LIN {X 0,Y 572.94,Z 558.785,A -85,B 0,C 180,E1 -2249.297,E2 -2249.297} C_VEL
LIN {X 0,Y 572.938,Z 559,A -85,B 0,C 180,E1 -2250,E2 -2250} C_VEL
LIN {X 0,Y 572.946,Z 558.187,A -85,B 0,C 180,E1 -2251.405,E2 -2251.405} C_VEL
LIN {X 0,Y 572.938,Z 557.2,A -85,B 0,C 180,E1 -2252.109,E2 -2252.109} C_VEL
LIN {X 0,Y 572.959,Z 555.811,A -85,B 0,C 180,E1 -2252.812,E2 -2252.812} C_VEL
LIN {X 0,Y 573.014,Z 552.897,A -85,B 0,C 180,E1 -2253.868,E2 -2253.868} C_VEL
LIN {X 0,Y 572.963,Z 548.951,A -85,B 0,C 180,E1 -2254.925,E2 -2254.925} C_VEL
LIN {X 0,Y 573.068,Z 542.879,A -85,B 0,C 180,E1 -2256.16,E2 -2256.16} C_VEL
LIN {X 0,Y 573.119,Z 536.241,A -85,B 0,C 180,E1 -2257.22,E2 -2257.22} C_VEL
LIN {X 0,Y 573.192,Z 527.995,A -85,B 0,C 180,E1 -2258.283,E2 -2258.283} C_VEL
LIN {X 0,Y 573.319,Z 517.606,A -85,B 0,C 180,E1 -2259.347,E2 -2259.347} C_VEL
LIN {X 0,Y 573.43,Z 507.931,A -85,B 0,C 180,E1 -2260.147,E2 -2260.147} C_VEL
LIN {X 0,Y 573.549,Z 497.409,A -85,B 0,C 180,E1 -2260.854,E2 -2260.854} C_VEL
LIN {X 0,Y 573.652,Z 486.295,A -85,B 0,C 180,E1 -2261.447,E2 -2261.447} C_VEL
LIN {X 0,Y 573.719,Z 473.186,A -85,B 0,C 180,E1 -2261.974,E2 -2261.974} C_VEL
LIN {X 0,Y 573.813,Z 460.539,A -85,B 0,C 180,E1 -2262.331,E2 -2262.331} C_VEL
LIN {X 0,Y 573.908,Z 447.35,A -85,B 0,C 180,E1 -2262.554,E2 -2262.554} C_VEL
LIN {X 0,Y 573.909,Z 350.315,A -85,B 0,C 180,E1 -2263.775,E2 -2263.775} C_VEL
LIN {X 0,Y 573.398,Z 346.617,A -85,B 0,C 180,E1 -2263.85,E2 -2263.85} C_VEL
LIN {X 0,Y 573.568,Z 326.123,A -85,B 0,C 180,E1 -2266.727,E2 -2266.727} C_VEL
LIN {X 0,Y 573.802,Z 305.615,A -85,B 0,C 180,E1 -2269.646,E2 -2269.646} C_VEL
LIN {X 0,Y 574.043,Z 285.799,A -85,B 0,C 180,E1 -2272.494,E2 -2272.494} C_VEL
LIN {X 0,Y 573.587,Z 280.858,A -85,B 0,C 180,E1 -2273.226,E2 -2273.226} C_VEL
LIN {X 0,Y 573.268,Z 279.079,A -85,B 0,C 180,E1 -2273.519,E2 -2273.519} C_VEL
LIN {X 0,Y 573.26,Z 279.079,A -85,B 0,C 180,E1 -2276.189,E2 -2276.189} C_VEL
LIN {X 0,Y 573.238,Z 279.076,A -85,B 0,C 180,E1 -2278.564,E2 -2278.564} C_VEL
LIN {X 0,Y 573.225,Z 279.075,A -85,B 0,C 180,E1 -2280.993,E2 -2280.993} C_VEL
LIN {X 0,Y 573.261,Z 279.072,A -85,B 0,C 180,E1 -2283.523,E2 -2283.523} C_VEL
LIN {X 0,Y 573.212,Z 279.084,A -85,B 0,C 180,E1 -2286.051,E2 -2286.051} C_VEL
LIN {X 0,Y 573.239,Z 279.077,A -85,B 0,C 180,E1 -2288.701,E2 -2288.701} C_VEL
LIN {X 0,Y 573.251,Z 279.072,A -85,B 0,C 180,E1 -2291.595,E2 -2291.595} C_VEL
LIN {X 0,Y 573.232,Z 279.082,A -85,B 0,C 180,E1 -2294.333,E2 -2294.333} C_VEL
LIN {X 0,Y 573.237,Z 279.074,A -85,B 0,C 180,E1 -2297.358,E2 -2297.358} C_VEL
LIN {X 0,Y 573.243,Z 279.079,A -85,B 0,C 180,E1 -2300.392,E2 -2300.392} C_VEL
LIN {X 0,Y 573.252,Z 279.076,A -85,B 0,C 180,E1 -2303.077,E2 -2303.077} C_VEL
LIN {X 0,Y 573.263,Z 279.07,A -85,B 0,C 180,E1 -2305.671,E2 -2305.671} C_VEL
LIN {X 0,Y 573.244,Z 279.074,A -85,B 0,C 180,E1 -2308.185,E2 -2308.185} C_VEL
LIN {X 0,Y 573.26,Z 279.076,A -85,B 0,C 180,E1 -2310.634,E2 -2310.634} C_VEL
LIN {X 0,Y 573.247,Z 279.083,A -85,B 0,C 180,E1 -2313.024,E2 -2313.024} C_VEL
LIN {X 0,Y 573.27,Z 279.075,A -85,B 0,C 180,E1 -2315.366,E2 -2315.366} C_VEL
LIN {X 0,Y 573.222,Z 279.076,A -85,B 0,C 180,E1 -2318.419,E2 -2318.419} C_VEL
LIN {X 0,Y 573.272,Z 279.072,A -85,B 0,C 180,E1 -2320.728,E2 -2320.728} C_VEL
LIN {X 0,Y 573.244,Z 279.077,A -85,B 0,C 180,E1 -2323.622,E2 -2323.622} C_VEL
LIN {X 0,Y 573.266,Z 279.073,A -85,B 0,C 180,E1 -2325.807,E2 -2325.807} C_VEL
LIN {X 0,Y 573.256,Z 279.072,A -85,B 0,C 180,E1 -2328.745,E2 -2328.745} C_VEL
LIN {X 0,Y 573.283,Z 279.078,A -85,B 0,C 180,E1 -2331.541,E2 -2331.541} C_VEL
LIN {X 0,Y 573.283,Z 279.068,A -85,B 0,C 180,E1 -2334.372,E2 -2334.372} C_VEL
LIN {X 0,Y 573.297,Z 279.073,A -85,B 0,C 180,E1 -2337.893,E2 -2337.893} C_VEL
LIN {X 0,Y 573.321,Z 279.063,A -85,B 0,C 180,E1 -2340.703,E2 -2340.703} C_VEL
LIN {X 0,Y 573.238,Z 279.079,A -85,B 0,C 180,E1 -2343.515,E2 -2343.515} C_VEL
LIN {X 0,Y 573.289,Z 279.073,A -85,B 0,C 180,E1 -2345.628,E2 -2345.628} C_VEL
LIN {X 0,Y 573.277,Z 279.071,A -85,B 0,C 180,E1 -2348.46,E2 -2348.46} C_VEL
LIN {X 0,Y 573.266,Z 279.071,A -85,B 0,C 180,E1 -2351.312,E2 -2351.312} C_VEL
LIN {X 0,Y 573.253,Z 279.081,A -85,B 0,C 180,E1 -2354.194,E2 -2354.194} C_VEL
LIN {X 0,Y 573.252,Z 279.072,A -85,B 0,C 180,E1 -2357.112,E2 -2357.112} C_VEL
LIN {X 0,Y 573.236,Z 279.081,A -85,B 0,C 180,E1 -2360.078,E2 -2360.078} C_VEL
LIN {X 0,Y 573.228,Z 279.086,A -85,B 0,C 180,E1 -2362.338,E2 -2362.338} C_VEL
LIN {X 0,Y 573.241,Z 279.077,A -85,B 0,C 180,E1 -2364.37,E2 -2364.37} C_VEL
LIN {X 0,Y 572.61,Z 279.158,A -85,B 0,C 180,E1 -2364.956,E2 -2364.956} C_VEL
LIN {X 0,Y 569.752,Z 279.513,A -85,B 0,C 180,E1 -2365.907,E2 -2365.907} C_VEL
LIN {X 0,Y 567.308,Z 279.819,A -85,B 0,C 180,E1 -2366.673,E2 -2366.673} C_VEL
LIN {X 0,Y 566.252,Z 279.944,A -85,B 0,C 180,E1 -2367.264,E2 -2367.264} C_VEL
LIN {X 0,Y 566.163,Z 279.955,A -85,B 0,C 180,E1 -2367.464,E2 -2367.464} C_VEL
LIN {X 0,Y 566.195,Z 279.951,A -85,B 0,C 180,E1 -2369.77,E2 -2369.77} C_VEL
LIN {X 0,Y 566.2,Z 279.958,A -85,B 0,C 180,E1 -2372.431,E2 -2372.431} C_VEL
LIN {X 0,Y 566.175,Z 279.958,A -85,B 0,C 180,E1 -2374.99,E2 -2374.99} C_VEL
LIN {X 0,Y 566.192,Z 279.952,A -85,B 0,C 180,E1 -2377.462,E2 -2377.462} C_VEL
LIN {X 0,Y 566.203,Z 279.951,A -85,B 0,C 180,E1 -2380.2,E2 -2380.2} C_VEL
LIN {X 0,Y 566.186,Z 279.96,A -85,B 0,C 180,E1 -2383.056,E2 -2383.056} C_VEL
LIN {X 0,Y 566.191,Z 279.951,A -85,B 0,C 180,E1 -2386.05,E2 -2386.05} C_VEL
LIN {X 0,Y 566.201,Z 279.958,A -85,B 0,C 180,E1 -2389.216,E2 -2389.216} C_VEL
LIN {X 0,Y 566.178,Z 279.956,A -85,B 0,C 180,E1 -2391.637,E2 -2391.637} C_VEL
LIN {X 0,Y 566.149,Z 279.956,A -85,B 0,C 180,E1 -2394.308,E2 -2394.308} C_VEL
LIN {X 0,Y 566.195,Z 279.955,A -85,B 0,C 180,E1 -2396.897,E2 -2396.897} C_VEL
LIN {X 0,Y 566.163,Z 279.964,A -85,B 0,C 180,E1 -2399.407,E2 -2399.407} C_VEL
LIN {X 0,Y 566.171,Z 279.957,A -85,B 0,C 180,E1 -2401.856,E2 -2401.856} C_VEL
LIN {X 0,Y 566.174,Z 279.954,A -85,B 0,C 180,E1 -2404.25,E2 -2404.25} C_VEL
LIN {X 0,Y 566.176,Z 279.96,A -85,B 0,C 180,E1 -2407.369,E2 -2407.369} C_VEL
LIN {X 0,Y 566.205,Z 279.96,A -85,B 0,C 180,E1 -2409.663,E2 -2409.663} C_VEL
LIN {X 0,Y 566.198,Z 279.951,A -85,B 0,C 180,E1 -2412.898,E2 -2412.898} C_VEL
LIN {X 0,Y 566.232,Z 279.954,A -85,B 0,C 180,E1 -2415.627,E2 -2415.627} C_VEL
LIN {X 0,Y 566.194,Z 279.951,A -85,B 0,C 180,E1 -2418.7,E2 -2418.7} C_VEL
LIN {X 0,Y 566.19,Z 279.954,A -85,B 0,C 180,E1 -2421.434,E2 -2421.434} C_VEL
LIN {X 0,Y 566.234,Z 279.952,A -85,B 0,C 180,E1 -2424.302,E2 -2424.302} C_VEL
LIN {X 0,Y 566.279,Z 279.947,A -85,B 0,C 180,E1 -2427.867,E2 -2427.867} C_VEL
LIN {X 0,Y 566.288,Z 279.947,A -85,B 0,C 180,E1 -2430,E2 -2430} C_VEL
LIN {X 0,Y 566.24,Z 279.947,A -85,B 0,C 180,E1 -2432.846,E2 -2432.846} C_VEL
LIN {X 0,Y 566.224,Z 279.948,A -85,B 0,C 180,E1 -2435.699,E2 -2435.699} C_VEL
LIN {X 0,Y 566.185,Z 279.96,A -85,B 0,C 180,E1 -2438.567,E2 -2438.567} C_VEL
LIN {X 0,Y 566.162,Z 279.955,A -85,B 0,C 180,E1 -2441.456,E2 -2441.456} C_VEL
LIN {X 0,Y 566.18,Z 279.962,A -85,B 0,C 180,E1 -2444.482,E2 -2444.482} C_VEL
LIN {X 0,Y 566.173,Z 279.954,A -85,B 0,C 180,E1 -2447.333,E2 -2447.333} C_VEL
LIN {X 0,Y 566.175,Z 279.953,A -85,B 0,C 180,E1 -2449.582,E2 -2449.582} C_VEL
LIN {X 0,Y 566.151,Z 279.957,A -85,B 0,C 180,E1 -2451.865,E2 -2451.865} C_VEL
LIN {X 0,Y 566.145,Z 279.96,A -85,B 0,C 180,E1 -2454.183,E2 -2454.183} C_VEL
LIN {X 0,Y 566.152,Z 279.964,A -85,B 0,C 180,E1 -2456.647,E2 -2456.647} C_VEL
LIN {X 0,Y 566.155,Z 279.966,A -85,B 0,C 180,E1 -2457.844,E2 -2457.844} C_VEL
LIN {X 0,Y 566.475,Z 284.764,A -85,B 0,C 180,E1 -2458.741,E2 -2458.741} C_VEL
LIN {X 0,Y 566.312,Z 299.374,A -85,B 0,C 180,E1 -2461.415,E2 -2461.415} C_VEL
LIN {X 0,Y 566.197,Z 308.432,A -85,B 0,C 180,E1 -2463.054,E2 -2463.054} C_VEL
LIN {X 0,Y 567.12,Z 313.95,A -85,B 0,C 180,E1 -2463.148,E2 -2463.148} C_VEL
LIN {X 0,Y 566.975,Z 415.264,A -85,B 0,C 180,E1 -2464.454,E2 -2464.454} C_VEL
LIN {X 0,Y 566.835,Z 428.571,A -85,B 0,C 180,E1 -2464.774,E2 -2464.774} C_VEL
LIN {X 0,Y 566.731,Z 439.996,A -85,B 0,C 180,E1 -2465.181,E2 -2465.181} C_VEL
LIN {X 0,Y 566.598,Z 450.313,A -85,B 0,C 180,E1 -2465.661,E2 -2465.661} C_VEL
LIN {X 0,Y 566.503,Z 460.478,A -85,B 0,C 180,E1 -2466.255,E2 -2466.255} C_VEL
LIN {X 0,Y 566.359,Z 469.422,A -85,B 0,C 180,E1 -2466.891,E2 -2466.891} C_VEL
LIN {X 0,Y 566.251,Z 477.431,A -85,B 0,C 180,E1 -2467.569,E2 -2467.569} C_VEL
LIN {X 0,Y 566.164,Z 485.34,A -85,B 0,C 180,E1 -2468.365,E2 -2468.365} C_VEL
LIN {X 0,Y 566.068,Z 492.963,A -85,B 0,C 180,E1 -2469.286,E2 -2469.286} C_VEL
LIN {X 0,Y 565.979,Z 499.365,A -85,B 0,C 180,E1 -2470.219,E2 -2470.219} C_VEL
LIN {X 0,Y 565.956,Z 504.694,A -85,B 0,C 180,E1 -2471.159,E2 -2471.159} C_VEL
LIN {X 0,Y 565.94,Z 509.114,A -85,B 0,C 180,E1 -2472.113,E2 -2472.113} C_VEL
LIN {X 0,Y 565.897,Z 512.699,A -85,B 0,C 180,E1 -2473.083,E2 -2473.083} C_VEL
LIN {X 0,Y 565.874,Z 515.471,A -85,B 0,C 180,E1 -2474.068,E2 -2474.068} C_VEL
LIN {X 0,Y 565.845,Z 517.452,A -85,B 0,C 180,E1 -2475.069,E2 -2475.069} C_VEL
LIN {X 0,Y 565.854,Z 518.623,A -85,B 0,C 180,E1 -2476.085,E2 -2476.085} C_VEL
LIN {X 0,Y 565.861,Z 518.99,A -85,B 0,C 180,E1 -2477.12,E2 -2477.12} C_VEL
LIN {X 0,Y 565.863,Z 518.499,A -85,B 0,C 180,E1 -2478.176,E2 -2478.176} C_VEL
LIN {X 0,Y 565.839,Z 517.081,A -85,B 0,C 180,E1 -2479.258,E2 -2479.258} C_VEL
LIN {X 0,Y 565.864,Z 513.657,A -85,B 0,C 180,E1 -2480.697,E2 -2480.697} C_VEL
LIN {X 0,Y 565.914,Z 510.584,A -85,B 0,C 180,E1 -2481.615,E2 -2481.615} C_VEL
LIN {X 0,Y 565.941,Z 506.208,A -85,B 0,C 180,E1 -2482.633,E2 -2482.633} C_VEL
LIN {X 0,Y 566.015,Z 500.789,A -85,B 0,C 180,E1 -2483.642,E2 -2483.642} C_VEL
LIN {X 0,Y 566.035,Z 493.84,A -85,B 0,C 180,E1 -2484.687,E2 -2484.687} C_VEL
LIN {X 0,Y 566.147,Z 486.369,A -85,B 0,C 180,E1 -2485.609,E2 -2485.609} C_VEL
LIN {X 0,Y 566.267,Z 477.878,A -85,B 0,C 180,E1 -2486.479,E2 -2486.479} C_VEL
LIN {X 0,Y 566.346,Z 468.29,A -85,B 0,C 180,E1 -2487.289,E2 -2487.289} C_VEL
LIN {X 0,Y 566.531,Z 456.725,A -85,B 0,C 180,E1 -2488.077,E2 -2488.077} C_VEL
LIN {X 0,Y 566.659,Z 445.1,A -85,B 0,C 180,E1 -2488.689,E2 -2488.689} C_VEL
LIN {X 0,Y 566.783,Z 433.171,A -85,B 0,C 180,E1 -2489.164,E2 -2489.164} C_VEL
LIN {X 0,Y 566.838,Z 422.732,A -85,B 0,C 180,E1 -2489.472,E2 -2489.472} C_VEL
LIN {X 0,Y 566.928,Z 410.787,A -85,B 0,C 180,E1 -2489.708,E2 -2489.708} C_VEL
LIN {X 0,Y 567.115,Z 313.681,A -85,B 0,C 180,E1 -2490.946,E2 -2490.946} C_VEL
LIN {X 0,Y 566.181,Z 308.374,A -85,B 0,C 180,E1 -2491.046,E2 -2491.046} C_VEL
LIN {X 0,Y 566.333,Z 295.048,A -85,B 0,C 180,E1 -2493.464,E2 -2493.464} C_VEL
LIN {X 0,Y 566.44,Z 282.076,A -85,B 0,C 180,E1 -2495.83,E2 -2495.83} C_VEL
LIN {X 0,Y 566.233,Z 279.951,A -85,B 0,C 180,E1 -2496.21,E2 -2496.21} C_VEL
LIN {X 0,Y 566.211,Z 279.955,A -85,B 0,C 180,E1 -2498.902,E2 -2498.902} C_VEL
LIN {X 0,Y 566.201,Z 279.959,A -85,B 0,C 180,E1 -2501.172,E2 -2501.172} C_VEL
LIN {X 0,Y 566.215,Z 279.96,A -85,B 0,C 180,E1 -2503.412,E2 -2503.412} C_VEL
LIN {X 0,Y 566.197,Z 279.952,A -85,B 0,C 180,E1 -2506.359,E2 -2506.359} C_VEL
LIN {X 0,Y 566.237,Z 279.946,A -85,B 0,C 180,E1 -2508.675,E2 -2508.675} C_VEL
LIN {X 0,Y 566.208,Z 279.957,A -85,B 0,C 180,E1 -2511.434,E2 -2511.434} C_VEL
LIN {X 0,Y 566.256,Z 279.946,A -85,B 0,C 180,E1 -2514.301,E2 -2514.301} C_VEL
LIN {X 0,Y 566.279,Z 279.951,A -85,B 0,C 180,E1 -2517.866,E2 -2517.866} C_VEL
LIN {X 0,Y 566.299,Z 279.938,A -85,B 0,C 180,E1 -2520.711,E2 -2520.711} C_VEL
LIN {X 0,Y 566.269,Z 279.942,A -85,B 0,C 180,E1 -2522.845,E2 -2522.845} C_VEL
LIN {X 0,Y 566.255,Z 279.947,A -85,B 0,C 180,E1 -2525.698,E2 -2525.698} C_VEL
LIN {X 0,Y 566.227,Z 279.951,A -85,B 0,C 180,E1 -2528.566,E2 -2528.566} C_VEL
LIN {X 0,Y 566.244,Z 279.945,A -85,B 0,C 180,E1 -2531.454,E2 -2531.454} C_VEL
LIN {X 0,Y 566.236,Z 279.955,A -85,B 0,C 180,E1 -2534.506,E2 -2534.506} C_VEL
LIN {X 0,Y 566.2,Z 279.949,A -85,B 0,C 180,E1 -2537.332,E2 -2537.332} C_VEL
LIN {X 0,Y 566.209,Z 279.956,A -85,B 0,C 180,E1 -2540.337,E2 -2540.337} C_VEL
LIN {X 0,Y 566.171,Z 279.955,A -85,B 0,C 180,E1 -2543.281,E2 -2543.281} C_VEL
LIN {X 0,Y 566.214,Z 279.948,A -85,B 0,C 180,E1 -2545.749,E2 -2545.749} C_VEL
LIN {X 0,Y 566.204,Z 279.95,A -85,B 0,C 180,E1 -2548.202,E2 -2548.202} C_VEL
LIN {X 0,Y 566.192,Z 279.959,A -85,B 0,C 180,E1 -2551.076,E2 -2551.076} C_VEL
LIN {X 0,Y 566.198,Z 279.951,A -85,B 0,C 180,E1 -2553.732,E2 -2553.732} C_VEL
LIN {X 0,Y 566.201,Z 279.953,A -85,B 0,C 180,E1 -2556.57,E2 -2556.57} C_VEL
LIN {X 0,Y 566.216,Z 279.951,A -85,B 0,C 180,E1 -2559.686,E2 -2559.686} C_VEL
LIN {X 0,Y 566.203,Z 279.954,A -85,B 0,C 180,E1 -2562.917,E2 -2562.917} C_VEL
LIN {X 0,Y 566.196,Z 279.953,A -85,B 0,C 180,E1 -2566.049,E2 -2566.049} C_VEL
LIN {X 0,Y 566.206,Z 279.955,A -85,B 0,C 180,E1 -2569.215,E2 -2569.215} C_VEL
LIN {X 0,Y 566.187,Z 279.963,A -85,B 0,C 180,E1 -2571.637,E2 -2571.637} C_VEL
LIN {X 0,Y 566.164,Z 279.958,A -85,B 0,C 180,E1 -2574.308,E2 -2574.308} C_VEL
LIN {X 0,Y 566.207,Z 279.951,A -85,B 0,C 180,E1 -2576.897,E2 -2576.897} C_VEL
LIN {X 0,Y 566.183,Z 279.957,A -85,B 0,C 180,E1 -2579.407,E2 -2579.407} C_VEL
LIN {X 0,Y 566.198,Z 279.961,A -85,B 0,C 180,E1 -2581.856,E2 -2581.856} C_VEL
LIN {X 0,Y 566.211,Z 279.958,A -85,B 0,C 180,E1 -2584.251,E2 -2584.251} C_VEL
LIN {X 0,Y 566.228,Z 280.1,A -85,B 0,C 180,E1 -2586.452,E2 -2586.452} C_VEL
LIN {X 0,Y 566.988,Z 285.18,A -85,B 0,C 180,E1 -2587.21,E2 -2587.21} C_VEL
LIN {X 0,Y 566.869,Z 303.894,A -85,B 0,C 180,E1 -2589.876,E2 -2589.876} C_VEL
LIN {X 0,Y 566.611,Z 324.89,A -85,B 0,C 180,E1 -2592.885,E2 -2592.885} C_VEL
LIN {X 0,Y 566.39,Z 346.61,A -85,B 0,C 180,E1 -2595.974,E2 -2595.974} C_VEL
LIN {X 0,Y 567.195,Z 353.264,A -85,B 0,C 180,E1 -2596.096,E2 -2596.096} C_VEL
LIN {X 0,Y 566.954,Z 454.929,A -85,B 0,C 180,E1 -2597.403,E2 -2597.403} C_VEL
LIN {X 0,Y 566.847,Z 467.445,A -85,B 0,C 180,E1 -2597.696,E2 -2597.696} C_VEL
LIN {X 0,Y 566.724,Z 480.368,A -85,B 0,C 180,E1 -2598.147,E2 -2598.147} C_VEL
LIN {X 0,Y 566.631,Z 492.042,A -85,B 0,C 180,E1 -2598.702,E2 -2598.702} C_VEL
LIN {X 0,Y 566.488,Z 502.902,A -85,B 0,C 180,E1 -2599.365,E2 -2599.365} C_VEL
LIN {X 0,Y 566.33,Z 513.535,A -85,B 0,C 180,E1 -2600.175,E2 -2600.175} C_VEL
LIN {X 0,Y 566.206,Z 523.08,A -85,B 0,C 180,E1 -2601.074,E2 -2601.074} C_VEL
LIN {X 0,Y 566.111,Z 530.958,A -85,B 0,C 180,E1 -2601.971,E2 -2601.971} C_VEL
LIN {X 0,Y 566.004,Z 538.62,A -85,B 0,C 180,E1 -2603.046,E2 -2603.046} C_VEL
LIN {X 0,Y 566.004,Z 545.678,A -85,B 0,C 180,E1 -2604.299,E2 -2604.299} C_VEL
LIN {X 0,Y 565.933,Z 550.371,A -85,B 0,C 180,E1 -2605.37,E2 -2605.37} C_VEL
LIN {X 0,Y 565.927,Z 553.957,A -85,B 0,C 180,E1 -2606.44,E2 -2606.44} C_VEL
LIN {X 0,Y 565.878,Z 555.807,A -85,B 0,C 180,E1 -2607.152,E2 -2607.152} C_VEL
LIN {X 0,Y 565.845,Z 558.184,A -85,B 0,C 180,E1 -2608.576,E2 -2608.576} C_VEL
LIN {X 0,Y 565.839,Z 559,A -85,B 0,C 180,E1 -2610,E2 -2610} C_VEL
LIN {X 0,Y 565.845,Z 558.186,A -85,B 0,C 180,E1 -2611.423,E2 -2611.423} C_VEL
LIN {X 0,Y 565.878,Z 555.811,A -85,B 0,C 180,E1 -2612.847,E2 -2612.847} C_VEL
LIN {X 0,Y 565.926,Z 552.897,A -85,B 0,C 180,E1 -2613.916,E2 -2613.916} C_VEL
LIN {X 0,Y 565.878,Z 548.951,A -85,B 0,C 180,E1 -2614.987,E2 -2614.987} C_VEL
LIN {X 0,Y 566.003,Z 543.869,A -85,B 0,C 180,E1 -2616.058,E2 -2616.058} C_VEL
LIN {X 0,Y 566.039,Z 537.471,A -85,B 0,C 180,E1 -2617.132,E2 -2617.132} C_VEL
LIN {X 0,Y 566.128,Z 529.482,A -85,B 0,C 180,E1 -2618.207,E2 -2618.207} C_VEL
LIN {X 0,Y 566.228,Z 521.34,A -85,B 0,C 180,E1 -2619.105,E2 -2619.105} C_VEL
LIN {X 0,Y 566.336,Z 511.406,A -85,B 0,C 180,E1 -2620.005,E2 -2620.005} C_VEL
LIN {X 0,Y 566.543,Z 500.309,A -85,B 0,C 180,E1 -2620.806,E2 -2620.806} C_VEL
LIN {X 0,Y 566.64,Z 489.184,A -85,B 0,C 180,E1 -2621.446,E2 -2621.446} C_VEL
LIN {X 0,Y 566.718,Z 476.994,A -85,B 0,C 180,E1 -2621.988,E2 -2621.988} C_VEL
LIN {X 0,Y 566.868,Z 464.196,A -85,B 0,C 180,E1 -2622.394,E2 -2622.394} C_VEL
LIN {X 0,Y 566.986,Z 450.635,A -85,B 0,C 180,E1 -2622.664,E2 -2622.664} C_VEL
LIN {X 0,Y 567.067,Z 351.208,A -85,B 0,C 180,E1 -2623.933,E2 -2623.933} C_VEL
LIN {X 0,Y 566.405,Z 346.617,A -85,B 0,C 180,E1 -2624.024,E2 -2624.024} C_VEL
LIN {X 0,Y 566.605,Z 324.044,A -85,B 0,C 180,E1 -2627.237,E2 -2627.237} C_VEL
LIN {X 0,Y 566.868,Z 303.978,A -85,B 0,C 180,E1 -2630.123,E2 -2630.123} C_VEL
LIN {X 0,Y 567.095,Z 285.582,A -85,B 0,C 180,E1 -2632.785,E2 -2632.785} C_VEL
LIN {X 0,Y 566.206,Z 279.96,A -85,B 0,C 180,E1 -2633.669,E2 -2633.669} C_VEL
LIN {X 0,Y 566.21,Z 279.958,A -85,B 0,C 180,E1 -2635.749,E2 -2635.749} C_VEL
LIN {X 0,Y 566.202,Z 279.958,A -85,B 0,C 180,E1 -2638.201,E2 -2638.201} C_VEL
LIN {X 0,Y 566.19,Z 279.951,A -85,B 0,C 180,E1 -2641.076,E2 -2641.076} C_VEL
LIN {X 0,Y 566.21,Z 279.952,A -85,B 0,C 180,E1 -2643.733,E2 -2643.733} C_VEL
LIN {X 0,Y 566.198,Z 279.956,A -85,B 0,C 180,E1 -2646.569,E2 -2646.569} C_VEL
LIN {X 0,Y 566.213,Z 279.95,A -85,B 0,C 180,E1 -2649.685,E2 -2649.685} C_VEL
LIN {X 0,Y 566.211,Z 279.954,A -85,B 0,C 180,E1 -2652.087,E2 -2652.087} C_VEL
LIN {X 0,Y 566.17,Z 279.956,A -85,B 0,C 180,E1 -2655.035,E2 -2655.035} C_VEL
LIN {X 0,Y 566.215,Z 279.952,A -85,B 0,C 180,E1 -2658.135,E2 -2658.135} C_VEL
LIN {X 0,Y 566.217,Z 279.958,A -85,B 0,C 180,E1 -2660.726,E2 -2660.726} C_VEL
LIN {X 0,Y 566.202,Z 279.95,A -85,B 0,C 180,E1 -2663.785,E2 -2663.785} C_VEL
LIN {X 0,Y 566.224,Z 279.957,A -85,B 0,C 180,E1 -2666.898,E2 -2666.898} C_VEL
LIN {X 0,Y 566.183,Z 279.955,A -85,B 0,C 180,E1 -2669.407,E2 -2669.407} C_VEL
LIN {X 0,Y 566.206,Z 279.949,A -85,B 0,C 180,E1 -2671.857,E2 -2671.857} C_VEL
LIN {X 0,Y 566.21,Z 279.949,A -85,B 0,C 180,E1 -2674.251,E2 -2674.251} C_VEL
LIN {X 0,Y 566.186,Z 279.956,A -85,B 0,C 180,E1 -2676.713,E2 -2676.713} C_VEL
LIN {X 0,Y 566.207,Z 279.952,A -85,B 0,C 180,E1 -2679.663,E2 -2679.663} C_VEL
LIN {X 0,Y 566.193,Z 279.953,A -85,B 0,C 180,E1 -2682.668,E2 -2682.668} C_VEL
LIN {X 0,Y 566.227,Z 279.952,A -85,B 0,C 180,E1 -2685.627,E2 -2685.627} C_VEL
LIN {X 0,Y 566.228,Z 279.947,A -85,B 0,C 180,E1 -2688.675,E2 -2688.675} C_VEL
LIN {X 0,Y 566.228,Z 279.957,A -85,B 0,C 180,E1 -2691.434,E2 -2691.434} C_VEL
LIN {X 0,Y 566.251,Z 279.944,A -85,B 0,C 180,E1 -2694.302,E2 -2694.302} C_VEL
LIN {X 0,Y 566.269,Z 279.949,A -85,B 0,C 180,E1 -2697.866,E2 -2697.866} C_VEL
LIN {X 0,Y 566.292,Z 279.939,A -85,B 0,C 180,E1 -2700.711,E2 -2700.711} C_VEL
LIN {X 0,Y 566.263,Z 279.942,A -85,B 0,C 180,E1 -2702.846,E2 -2702.846} C_VEL
LIN {X 0,Y 566.255,Z 279.951,A -85,B 0,C 180,E1 -2705.699,E2 -2705.699} C_VEL
LIN {X 0,Y 566.221,Z 279.949,A -85,B 0,C 180,E1 -2708.566,E2 -2708.566} C_VEL
LIN {X 0,Y 566.236,Z 279.947,A -85,B 0,C 180,E1 -2711.455,E2 -2711.455} C_VEL
LIN {X 0,Y 566.217,Z 279.952,A -85,B 0,C 180,E1 -2714.502,E2 -2714.502} C_VEL
LIN {X 0,Y 566.192,Z 279.951,A -85,B 0,C 180,E1 -2717.332,E2 -2717.332} C_VEL
LIN {X 0,Y 566.201,Z 279.96,A -85,B 0,C 180,E1 -2720.338,E2 -2720.338} C_VEL
LIN {X 0,Y 566.164,Z 279.955,A -85,B 0,C 180,E1 -2723.281,E2 -2723.281} C_VEL
LIN {X 0,Y 566.204,Z 279.951,A -85,B 0,C 180,E1 -2725.75,E2 -2725.75} C_VEL
LIN {X 0,Y 566.163,Z 279.955,A -85,B 0,C 180,E1 -2727.464,E2 -2727.464} C_VEL
LIN {X 0,Y 565.492,Z 280.043,A -85,B 0,C 180,E1 -2728.058,E2 -2728.058} C_VEL
LIN {X 0,Y 562.641,Z 280.396,A -85,B 0,C 180,E1 -2729.022,E2 -2729.022} C_VEL
LIN {X 0,Y 560.239,Z 280.695,A -85,B 0,C 180,E1 -2729.798,E2 -2729.798} C_VEL
LIN {X 0,Y 559.214,Z 280.828,A -85,B 0,C 180,E1 -2730.397,E2 -2730.397} C_VEL
LIN {X 0,Y 559.134,Z 280.832,A -85,B 0,C 180,E1 -2730.6,E2 -2730.6} C_VEL
LIN {X 0,Y 559.149,Z 280.837,A -85,B 0,C 180,E1 -2732.716,E2 -2732.716} C_VEL
LIN {X 0,Y 559.123,Z 280.833,A -85,B 0,C 180,E1 -2735.325,E2 -2735.325} C_VEL
LIN {X 0,Y 559.128,Z 280.832,A -85,B 0,C 180,E1 -2738.018,E2 -2738.018} C_VEL
LIN {X 0,Y 559.151,Z 280.839,A -85,B 0,C 180,E1 -2740.813,E2 -2740.813} C_VEL
LIN {X 0,Y 559.108,Z 280.834,A -85,B 0,C 180,E1 -2743.738,E2 -2743.738} C_VEL
LIN {X 0,Y 559.134,Z 280.831,A -85,B 0,C 180,E1 -2746.266,E2 -2746.266} C_VEL
LIN {X 0,Y 559.152,Z 280.837,A -85,B 0,C 180,E1 -2749.188,E2 -2749.188} C_VEL
LIN {X 0,Y 559.126,Z 280.831,A -85,B 0,C 180,E1 -2751.983,E2 -2751.983} C_VEL
LIN {X 0,Y 559.128,Z 280.835,A -85,B 0,C 180,E1 -2754.789,E2 -2754.789} C_VEL
LIN {X 0,Y 559.149,Z 280.838,A -85,B 0,C 180,E1 -2757.367,E2 -2757.367} C_VEL
LIN {X 0,Y 559.112,Z 280.834,A -85,B 0,C 180,E1 -2760.15,E2 -2760.15} C_VEL
LIN {X 0,Y 559.116,Z 280.839,A -85,B 0,C 180,E1 -2763.185,E2 -2763.185} C_VEL
LIN {X 0,Y 559.103,Z 280.845,A -85,B 0,C 180,E1 -2765.493,E2 -2765.493} C_VEL
LIN {X 0,Y 559.174,Z 280.825,A -85,B 0,C 180,E1 -2768.625,E2 -2768.625} C_VEL
LIN {X 0,Y 559.14,Z 280.83,A -85,B 0,C 180,E1 -2770.926,E2 -2770.926} C_VEL
LIN {X 0,Y 559.141,Z 280.836,A -85,B 0,C 180,E1 -2773.948,E2 -2773.948} C_VEL
LIN {X 0,Y 559.158,Z 280.831,A -85,B 0,C 180,E1 -2776.184,E2 -2776.184} C_VEL
LIN {X 0,Y 559.167,Z 280.827,A -85,B 0,C 180,E1 -2779.133,E2 -2779.133} C_VEL
LIN {X 0,Y 559.141,Z 280.839,A -85,B 0,C 180,E1 -2782.053,E2 -2782.053} C_VEL
LIN {X 0,Y 559.227,Z 280.819,A -85,B 0,C 180,E1 -2784.954,E2 -2784.954} C_VEL
LIN {X 0,Y 559.25,Z 280.822,A -85,B 0,C 180,E1 -2787.84,E2 -2787.84} C_VEL
LIN {X 0,Y 559.257,Z 280.823,A -85,B 0,C 180,E1 -2790,E2 -2790} C_VEL
LIN {X 0,Y 559.207,Z 280.823,A -85,B 0,C 180,E1 -2792.882,E2 -2792.882} C_VEL
LIN {X 0,Y 559.196,Z 280.825,A -85,B 0,C 180,E1 -2795.771,E2 -2795.771} C_VEL
LIN {X 0,Y 559.151,Z 280.834,A -85,B 0,C 180,E1 -2798.675,E2 -2798.675} C_VEL
LIN {X 0,Y 559.119,Z 280.832,A -85,B 0,C 180,E1 -2801.603,E2 -2801.603} C_VEL
LIN {X 0,Y 559.138,Z 280.841,A -85,B 0,C 180,E1 -2804.568,E2 -2804.568} C_VEL
LIN {X 0,Y 559.122,Z 280.832,A -85,B 0,C 180,E1 -2807.558,E2 -2807.558} C_VEL
LIN {X 0,Y 559.139,Z 280.83,A -85,B 0,C 180,E1 -2809.839,E2 -2809.839} C_VEL
LIN {X 0,Y 559.108,Z 280.836,A -85,B 0,C 180,E1 -2812.155,E2 -2812.155} C_VEL
LIN {X 0,Y 559.115,Z 280.84,A -85,B 0,C 180,E1 -2815.172,E2 -2815.172} C_VEL
LIN {X 0,Y 559.152,Z 280.838,A -85,B 0,C 180,E1 -2817.765,E2 -2817.765} C_VEL
LIN {X 0,Y 559.436,Z 287.057,A -85,B 0,C 180,E1 -2818.925,E2 -2818.925} C_VEL
LIN {X 0,Y 559.256,Z 301.165,A -85,B 0,C 180,E1 -2821.543,E2 -2821.543} C_VEL
LIN {X 0,Y 559.185,Z 308.337,A -85,B 0,C 180,E1 -2822.859,E2 -2822.859} C_VEL
LIN {X 0,Y 560.276,Z 315.962,A -85,B 0,C 180,E1 -2823.001,E2 -2823.001} C_VEL
LIN {X 0,Y 560.052,Z 414.689,A -85,B 0,C 180,E1 -2824.287,E2 -2824.287} C_VEL
LIN {X 0,Y 559.904,Z 428.248,A -85,B 0,C 180,E1 -2824.61,E2 -2824.61} C_VEL
LIN {X 0,Y 559.789,Z 439.278,A -85,B 0,C 180,E1 -2825.001,E2 -2825.001} C_VEL
LIN {X 0,Y 559.616,Z 450.392,A -85,B 0,C 180,E1 -2825.522,E2 -2825.522} C_VEL
LIN {X 0,Y 559.474,Z 459.651,A -85,B 0,C 180,E1 -2826.063,E2 -2826.063} C_VEL
LIN {X 0,Y 559.358,Z 469.295,A -85,B 0,C 180,E1 -2826.753,E2 -2826.753} C_VEL
LIN {X 0,Y 559.211,Z 478.012,A -85,B 0,C 180,E1 -2827.506,E2 -2827.506} C_VEL
LIN {X 0,Y 559.125,Z 485.261,A -85,B 0,C 180,E1 -2828.247,E2 -2828.247} C_VEL
LIN {X 0,Y 559.038,Z 491.164,A -85,B 0,C 180,E1 -2828.946,E2 -2828.946} C_VEL
LIN {X 0,Y 558.942,Z 498.017,A -85,B 0,C 180,E1 -2829.914,E2 -2829.914} C_VEL
LIN {X 0,Y 558.859,Z 504.336,A -85,B 0,C 180,E1 -2831.014,E2 -2831.014} C_VEL
LIN {X 0,Y 558.845,Z 509.302,A -85,B 0,C 180,E1 -2832.099,E2 -2832.099} C_VEL
LIN {X 0,Y 558.807,Z 513.074,A -85,B 0,C 180,E1 -2833.159,E2 -2833.159} C_VEL
LIN {X 0,Y 558.786,Z 515.827,A -85,B 0,C 180,E1 -2834.2,E2 -2834.2} C_VEL
LIN {X 0,Y 558.762,Z 517.673,A -85,B 0,C 180,E1 -2835.222,E2 -2835.222} C_VEL
LIN {X 0,Y 558.763,Z 518.703,A -85,B 0,C 180,E1 -2836.228,E2 -2836.228} C_VEL
LIN {X 0,Y 558.758,Z 518.969,A -85,B 0,C 180,E1 -2837.218,E2 -2837.218} C_VEL
LIN {X 0,Y 558.767,Z 518.496,A -85,B 0,C 180,E1 -2838.193,E2 -2838.193} C_VEL
LIN {X 0,Y 558.756,Z 517.29,A -85,B 0,C 180,E1 -2839.152,E2 -2839.152} C_VEL
LIN {X 0,Y 558.776,Z 514.168,A -85,B 0,C 180,E1 -2840.571,E2 -2840.571} C_VEL
LIN {X 0,Y 558.827,Z 510.862,A -85,B 0,C 180,E1 -2841.601,E2 -2841.601} C_VEL
LIN {X 0,Y 558.872,Z 506.538,A -85,B 0,C 180,E1 -2842.637,E2 -2842.637} C_VEL
LIN {X 0,Y 558.928,Z 500.49,A -85,B 0,C 180,E1 -2843.773,E2 -2843.773} C_VEL
LIN {X 0,Y 558.965,Z 494.719,A -85,B 0,C 180,E1 -2844.664,E2 -2844.664} C_VEL
LIN {X 0,Y 559.094,Z 487.826,A -85,B 0,C 180,E1 -2845.551,E2 -2845.551} C_VEL
LIN {X 0,Y 559.196,Z 479.658,A -85,B 0,C 180,E1 -2846.427,E2 -2846.427} C_VEL
LIN {X 0,Y 559.339,Z 471.129,A -85,B 0,C 180,E1 -2847.189,E2 -2847.189} C_VEL
LIN {X 0,Y 559.402,Z 462.547,A -85,B 0,C 180,E1 -2847.834,E2 -2847.834} C_VEL
LIN {X 0,Y 559.573,Z 453.655,A -85,B 0,C 180,E1 -2848.389,E2 -2848.389} C_VEL
LIN {X 0,Y 559.688,Z 444.104,A -85,B 0,C 180,E1 -2848.879,E2 -2848.879} C_VEL
LIN {X 0,Y 559.84,Z 434.109,A -85,B 0,C 180,E1 -2849.284,E2 -2849.284} C_VEL
LIN {X 0,Y 559.896,Z 423.293,A -85,B 0,C 180,E1 -2849.614,E2 -2849.614} C_VEL
LIN {X 0,Y 560.014,Z 412.313,A -85,B 0,C 180,E1 -2849.842,E2 -2849.842} C_VEL
LIN {X 0,Y 560.16,Z 314.154,A -85,B 0,C 180,E1 -2851.116,E2 -2851.116} C_VEL
LIN {X 0,Y 559.179,Z 308.486,A -85,B 0,C 180,E1 -2851.214,E2 -2851.214} C_VEL
LIN {X 0,Y 559.334,Z 294.686,A -85,B 0,C 180,E1 -2853.719,E2 -2853.719} C_VEL
LIN {X 0,Y 559.289,Z 281.037,A -85,B 0,C 180,E1 -2856.044,E2 -2856.044} C_VEL
LIN {X 0,Y 559.171,Z 280.832,A -85,B 0,C 180,E1 -2856.565,E2 -2856.565} C_VEL
LIN {X 0,Y 559.178,Z 280.835,A -85,B 0,C 180,E1 -2859.395,E2 -2859.395} C_VEL
LIN {X 0,Y 559.144,Z 280.836,A -85,B 0,C 180,E1 -2861.685,E2 -2861.685} C_VEL
LIN {X 0,Y 559.166,Z 280.831,A -85,B 0,C 180,E1 -2863.948,E2 -2863.948} C_VEL
LIN {X 0,Y 559.172,Z 280.828,A -85,B 0,C 180,E1 -2866.184,E2 -2866.184} C_VEL
LIN {X 0,Y 559.195,Z 280.827,A -85,B 0,C 180,E1 -2869.133,E2 -2869.133} C_VEL
LIN {X 0,Y 559.197,Z 280.828,A -85,B 0,C 180,E1 -2872.053,E2 -2872.053} C_VEL
LIN {X 0,Y 559.252,Z 280.817,A -85,B 0,C 180,E1 -2874.953,E2 -2874.953} C_VEL
LIN {X 0,Y 559.251,Z 280.826,A -85,B 0,C 180,E1 -2877.839,E2 -2877.839} C_VEL
LIN {X 0,Y 559.27,Z 280.813,A -85,B 0,C 180,E1 -2880.72,E2 -2880.72} C_VEL
LIN {X 0,Y 559.236,Z 280.818,A -85,B 0,C 180,E1 -2882.881,E2 -2882.881} C_VEL
LIN {X 0,Y 559.223,Z 280.824,A -85,B 0,C 180,E1 -2885.77,E2 -2885.77} C_VEL
LIN {X 0,Y 559.186,Z 280.827,A -85,B 0,C 180,E1 -2888.674,E2 -2888.674} C_VEL
LIN {X 0,Y 559.207,Z 280.822,A -85,B 0,C 180,E1 -2891.6,E2 -2891.6} C_VEL
LIN {X 0,Y 559.202,Z 280.83,A -85,B 0,C 180,E1 -2894.595,E2 -2894.595} C_VEL
LIN {X 0,Y 559.143,Z 280.828,A -85,B 0,C 180,E1 -2897.557,E2 -2897.557} C_VEL
LIN {X 0,Y 559.167,Z 280.827,A -85,B 0,C 180,E1 -2899.838,E2 -2899.838} C_VEL
LIN {X 0,Y 559.142,Z 280.832,A -85,B 0,C 180,E1 -2902.153,E2 -2902.153} C_VEL
LIN {X 0,Y 559.177,Z 280.827,A -85,B 0,C 180,E1 -2905.298,E2 -2905.298} C_VEL
LIN {X 0,Y 559.149,Z 280.827,A -85,B 0,C 180,E1 -2907.714,E2 -2907.714} C_VEL
LIN {X 0,Y 559.155,Z 280.829,A -85,B 0,C 180,E1 -2910.183,E2 -2910.183} C_VEL
LIN {X 0,Y 559.153,Z 280.833,A -85,B 0,C 180,E1 -2912.716,E2 -2912.716} C_VEL
LIN {X 0,Y 559.128,Z 280.838,A -85,B 0,C 180,E1 -2915.324,E2 -2915.324} C_VEL
LIN {X 0,Y 559.134,Z 280.83,A -85,B 0,C 180,E1 -2918.018,E2 -2918.018} C_VEL
LIN {X 0,Y 559.157,Z 280.831,A -85,B 0,C 180,E1 -2920.812,E2 -2920.812} C_VEL
LIN {X 0,Y 559.14,Z 280.834,A -85,B 0,C 180,E1 -2923.734,E2 -2923.734} C_VEL
LIN {X 0,Y 559.147,Z 280.831,A -85,B 0,C 180,E1 -2926.804,E2 -2926.804} C_VEL
LIN {X 0,Y 559.158,Z 280.833,A -85,B 0,C 180,E1 -2929.188,E2 -2929.188} C_VEL
LIN {X 0,Y 559.134,Z 280.836,A -85,B 0,C 180,E1 -2931.982,E2 -2931.982} C_VEL
LIN {X 0,Y 559.133,Z 280.832,A -85,B 0,C 180,E1 -2934.787,E2 -2934.787} C_VEL
LIN {X 0,Y 559.156,Z 280.833,A -85,B 0,C 180,E1 -2937.365,E2 -2937.365} C_VEL
LIN {X 0,Y 559.151,Z 280.836,A -85,B 0,C 180,E1 -2940.143,E2 -2940.143} C_VEL
LIN {X 0,Y 559.167,Z 280.829,A -85,B 0,C 180,E1 -2943.097,E2 -2943.097} C_VEL
LIN {X 0,Y 559.161,Z 280.833,A -85,B 0,C 180,E1 -2945.495,E2 -2945.495} C_VEL
LIN {X 0,Y 559.206,Z 280.932,A -85,B 0,C 180,E1 -2946.326,E2 -2946.326} C_VEL
LIN {X 0,Y 560.069,Z 287.396,A -85,B 0,C 180,E1 -2947.302,E2 -2947.302} C_VEL
LIN {X 0,Y 559.83,Z 309.025,A -85,B 0,C 180,E1 -2950.415,E2 -2950.415} C_VEL
LIN {X 0,Y 559.599,Z 328.65,A -85,B 0,C 180,E1 -2953.21,E2 -2953.21} C_VEL
LIN {X 0,Y 559.397,Z 346.61,A -85,B 0,C 180,E1 -2955.795,E2 -2955.795} C_VEL
LIN {X 0,Y 560.279,Z 354.271,A -85,B 0,C 180,E1 -2955.934,E2 -2955.934} C_VEL
LIN {X 0,Y 560.024,Z 454.929,A -85,B 0,C 180,E1 -2957.244,E2 -2957.244} C_VEL
LIN {X 0,Y 559.915,Z 468.206,A -85,B 0,C 180,E1 -2957.564,E2 -2957.564} C_VEL
LIN {X 0,Y 559.797,Z 480.369,A -85,B 0,C 180,E1 -2957.999,E2 -2957.999} C_VEL
LIN {X 0,Y 559.669,Z 491.803,A -85,B 0,C 180,E1 -2958.547,E2 -2958.547} C_VEL
LIN {X 0,Y 559.505,Z 502.9,A -85,B 0,C 180,E1 -2959.231,E2 -2959.231} C_VEL
LIN {X 0,Y 559.309,Z 513.534,A -85,B 0,C 180,E1 -2960.05,E2 -2960.05} C_VEL
LIN {X 0,Y 559.161,Z 523.093,A -85,B 0,C 180,E1 -2960.96,E2 -2960.96} C_VEL
LIN {X 0,Y 559.047,Z 530.958,A -85,B 0,C 180,E1 -2961.869,E2 -2961.869} C_VEL
LIN {X 0,Y 558.944,Z 538.62,A -85,B 0,C 180,E1 -2962.958,E2 -2962.958} C_VEL
LIN {X 0,Y 558.936,Z 545.678,A -85,B 0,C 180,E1 -2964.226,E2 -2964.226} C_VEL
LIN {X 0,Y 558.826,Z 550.371,A -85,B 0,C 180,E1 -2965.311,E2 -2965.311} C_VEL
LIN {X 0,Y 558.836,Z 553.957,A -85,B 0,C 180,E1 -2966.394,E2 -2966.394} C_VEL
LIN {X 0,Y 558.799,Z 555.807,A -85,B 0,C 180,E1 -2967.116,E2 -2967.116} C_VEL
LIN {X 0,Y 558.745,Z 558.183,A -85,B 0,C 180,E1 -2968.558,E2 -2968.558} C_VEL
LIN {X 0,Y 558.74,Z 559,A -85,B 0,C 180,E1 -2970,E2 -2970} C_VEL
LIN {X 0,Y 558.745,Z 558.185,A -85,B 0,C 180,E1 -2971.441,E2 -2971.441} C_VEL
LIN {X 0,Y 558.799,Z 555.811,A -85,B 0,C 180,E1 -2972.883,E2 -2972.883} C_VEL
LIN {X 0,Y 558.843,Z 552.897,A -85,B 0,C 180,E1 -2973.966,E2 -2973.966} C_VEL
LIN {X 0,Y 558.798,Z 548.95,A -85,B 0,C 180,E1 -2975.05,E2 -2975.05} C_VEL
LIN {X 0,Y 558.92,Z 543.87,A -85,B 0,C 180,E1 -2976.135,E2 -2976.135} C_VEL
LIN {X 0,Y 558.976,Z 537.471,A -85,B 0,C 180,E1 -2977.222,E2 -2977.222} C_VEL
LIN {X 0,Y 559.091,Z 529.481,A -85,B 0,C 180,E1 -2978.311,E2 -2978.311} C_VEL
LIN {X 0,Y 559.184,Z 521.339,A -85,B 0,C 180,E1 -2979.221,E2 -2979.221} C_VEL
LIN {X 0,Y 559.346,Z 511.405,A -85,B 0,C 180,E1 -2980.131,E2 -2980.131} C_VEL
LIN {X 0,Y 559.569,Z 500.387,A -85,B 0,C 180,E1 -2980.937,E2 -2980.937} C_VEL
LIN {X 0,Y 559.67,Z 488.469,A -85,B 0,C 180,E1 -2981.627,E2 -2981.627} C_VEL
LIN {X 0,Y 559.813,Z 475.782,A -85,B 0,C 180,E1 -2982.184,E2 -2982.184} C_VEL
LIN {X 0,Y 559.926,Z 462.366,A -85,B 0,C 180,E1 -2982.596,E2 -2982.596} C_VEL
LIN {X 0,Y 560.097,Z 449.121,A -85,B 0,C 180,E1 -2982.846,E2 -2982.846} C_VEL
LIN {X 0,Y 560.223,Z 352.325,A -85,B 0,C 180,E1 -2984.093,E2 -2984.093} C_VEL
LIN {X 0,Y 559.408,Z 346.617,A -85,B 0,C 180,E1 -2984.204,E2 -2984.204} C_VEL
LIN {X 0,Y 559.617,Z 324.701,A -85,B 0,C 180,E1 -2987.359,E2 -2987.359} C_VEL
LIN {X 0,Y 559.887,Z 306.388,A -85,B 0,C 180,E1 -2990.002,E2 -2990.002} C_VEL
LIN {X 0,Y 560.175,Z 287.997,A -85,B 0,C 180,E1 -2992.692,E2 -2992.692} C_VEL
LIN {X 0,Y 559.864,Z 284.509,A -85,B 0,C 180,E1 -2993.225,E2 -2993.225} C_VEL
LIN {X 0,Y 559.187,Z 280.835,A -85,B 0,C 180,E1 -2993.812,E2 -2993.812} C_VEL
LIN {X 0,Y 559.17,Z 280.828,A -85,B 0,C 180,E1 -2996.827,E2 -2996.827} C_VEL
LIN {X 0,Y 559.142,Z 280.831,A -85,B 0,C 180,E1 -2999.353,E2 -2999.353} C_VEL
LIN {X 0,Y 559.164,Z 280.832,A -85,B 0,C 180,E1 -3001.862,E2 -3001.862} C_VEL
LIN {X 0,Y 559.142,Z 280.836,A -85,B 0,C 180,E1 -3004.444,E2 -3004.444} C_VEL
LIN {X 0,Y 559.138,Z 280.83,A -85,B 0,C 180,E1 -3007.108,E2 -3007.108} C_VEL
LIN {X 0,Y 559.158,Z 280.831,A -85,B 0,C 180,E1 -3009.941,E2 -3009.941} C_VEL
LIN {X 0,Y 559.159,Z 280.832,A -85,B 0,C 180,E1 -3012.743,E2 -3012.743} C_VEL
LIN {X 0,Y 559.15,Z 280.829,A -85,B 0,C 180,E1 -3015.76,E2 -3015.76} C_VEL
LIN {X 0,Y 559.188,Z 280.828,A -85,B 0,C 180,E1 -3018.232,E2 -3018.232} C_VEL
LIN {X 0,Y 559.174,Z 280.828,A -85,B 0,C 180,E1 -3021.191,E2 -3021.191} C_VEL
LIN {X 0,Y 559.157,Z 280.827,A -85,B 0,C 180,E1 -3023.79,E2 -3023.79} C_VEL
LIN {X 0,Y 559.16,Z 280.831,A -85,B 0,C 180,E1 -3026.425,E2 -3026.425} C_VEL
LIN {X 0,Y 559.159,Z 280.836,A -85,B 0,C 180,E1 -3028.981,E2 -3028.981} C_VEL
LIN {X 0,Y 559.163,Z 280.828,A -85,B 0,C 180,E1 -3031.618,E2 -3031.618} C_VEL
LIN {X 0,Y 559.177,Z 280.825,A -85,B 0,C 180,E1 -3033.903,E2 -3033.903} C_VEL
LIN {X 0,Y 559.151,Z 280.831,A -85,B 0,C 180,E1 -3036.567,E2 -3036.567} C_VEL
LIN {X 0,Y 559.174,Z 280.832,A -85,B 0,C 180,E1 -3039.395,E2 -3039.395} C_VEL
LIN {X 0,Y 559.141,Z 280.833,A -85,B 0,C 180,E1 -3041.686,E2 -3041.686} C_VEL
LIN {X 0,Y 559.16,Z 280.828,A -85,B 0,C 180,E1 -3043.948,E2 -3043.948} C_VEL
LIN {X 0,Y 559.167,Z 280.826,A -85,B 0,C 180,E1 -3046.184,E2 -3046.184} C_VEL
LIN {X 0,Y 559.188,Z 280.829,A -85,B 0,C 180,E1 -3049.133,E2 -3049.133} C_VEL
LIN {X 0,Y 559.201,Z 280.824,A -85,B 0,C 180,E1 -3052.054,E2 -3052.054} C_VEL
LIN {X 0,Y 559.25,Z 280.817,A -85,B 0,C 180,E1 -3054.953,E2 -3054.953} C_VEL
LIN {X 0,Y 559.241,Z 280.824,A -85,B 0,C 180,E1 -3057.84,E2 -3057.84} C_VEL
LIN {X 0,Y 559.263,Z 280.814,A -85,B 0,C 180,E1 -3060.72,E2 -3060.72} C_VEL
LIN {X 0,Y 559.23,Z 280.818,A -85,B 0,C 180,E1 -3062.882,E2 -3062.882} C_VEL
LIN {X 0,Y 559.223,Z 280.828,A -85,B 0,C 180,E1 -3065.77,E2 -3065.77} C_VEL
LIN {X 0,Y 559.18,Z 280.825,A -85,B 0,C 180,E1 -3068.675,E2 -3068.675} C_VEL
LIN {X 0,Y 559.2,Z 280.826,A -85,B 0,C 180,E1 -3071.601,E2 -3071.601} C_VEL
LIN {X 0,Y 559.175,Z 280.828,A -85,B 0,C 180,E1 -3074.588,E2 -3074.588} C_VEL
LIN {X 0,Y 559.135,Z 280.832,A -85,B 0,C 180,E1 -3077.558,E2 -3077.558} C_VEL
LIN {X 0,Y 559.16,Z 280.831,A -85,B 0,C 180,E1 -3079.838,E2 -3079.838} C_VEL
LIN {X 0,Y 559.135,Z 280.838,A -85,B 0,C 180,E1 -3082.153,E2 -3082.153} C_VEL
LIN {X 0,Y 559.17,Z 280.826,A -85,B 0,C 180,E1 -3085.299,E2 -3085.299} C_VEL
LIN {X 0,Y 559.123,Z 280.832,A -85,B 0,C 180,E1 -3087.716,E2 -3087.716} C_VEL
LIN {X 0,Y 559.134,Z 280.832,A -85,B 0,C 180,E1 -3090.6,E2 -3090.6} C_VEL
LIN {X 0,Y 558.471,Z 280.916,A -85,B 0,C 180,E1 -3091.201,E2 -3091.201} C_VEL
LIN {X 0,Y 555.608,Z 281.273,A -85,B 0,C 180,E1 -3092.177,E2 -3092.177} C_VEL
LIN {X 0,Y 553.197,Z 281.575,A -85,B 0,C 180,E1 -3092.963,E2 -3092.963} C_VEL
LIN {X 0,Y 552.178,Z 281.697,A -85,B 0,C 180,E1 -3093.569,E2 -3093.569} C_VEL
LIN {X 0,Y 552.104,Z 281.706,A -85,B 0,C 180,E1 -3093.775,E2 -3093.775} C_VEL
LIN {X 0,Y 552.102,Z 281.717,A -85,B 0,C 180,E1 -3096.748,E2 -3096.748} C_VEL
LIN {X 0,Y 552.125,Z 281.704,A -85,B 0,C 180,E1 -3099.528,E2 -3099.528} C_VEL
LIN {X 0,Y 552.107,Z 281.709,A -85,B 0,C 180,E1 -3102.428,E2 -3102.428} C_VEL
LIN {X 0,Y 552.089,Z 281.71,A -85,B 0,C 180,E1 -3105.563,E2 -3105.563} C_VEL
LIN {X 0,Y 552.074,Z 281.713,A -85,B 0,C 180,E1 -3108.551,E2 -3108.551} C_VEL
LIN {X 0,Y 552.112,Z 281.711,A -85,B 0,C 180,E1 -3111.411,E2 -3111.411} C_VEL
LIN {X 0,Y 552.074,Z 281.71,A -85,B 0,C 180,E1 -3114.156,E2 -3114.156} C_VEL
LIN {X 0,Y 552.104,Z 281.709,A -85,B 0,C 180,E1 -3116.814,E2 -3116.814} C_VEL
LIN {X 0,Y 552.089,Z 281.718,A -85,B 0,C 180,E1 -3119.391,E2 -3119.391} C_VEL
LIN {X 0,Y 552.061,Z 281.714,A -85,B 0,C 180,E1 -3121.9,E2 -3121.9} C_VEL
LIN {X 0,Y 552.08,Z 281.709,A -85,B 0,C 180,E1 -3124.668,E2 -3124.668} C_VEL
LIN {X 0,Y 552.091,Z 281.718,A -85,B 0,C 180,E1 -3127.55,E2 -3127.55} C_VEL
LIN {X 0,Y 552.118,Z 281.705,A -85,B 0,C 180,E1 -3130.384,E2 -3130.384} C_VEL
LIN {X 0,Y 552.109,Z 281.706,A -85,B 0,C 180,E1 -3132.976,E2 -3132.976} C_VEL
LIN {X 0,Y 552.127,Z 281.71,A -85,B 0,C 180,E1 -3136.005,E2 -3136.005} C_VEL
LIN {X 0,Y 552.128,Z 281.703,A -85,B 0,C 180,E1 -3138.993,E2 -3138.993} C_VEL
LIN {X 0,Y 552.11,Z 281.716,A -85,B 0,C 180,E1 -3141.951,E2 -3141.951} C_VEL
LIN {X 0,Y 552.204,Z 281.694,A -85,B 0,C 180,E1 -3144.889,E2 -3144.889} C_VEL
LIN {X 0,Y 552.221,Z 281.697,A -85,B 0,C 180,E1 -3147.812,E2 -3147.812} C_VEL
LIN {X 0,Y 552.225,Z 281.698,A -85,B 0,C 180,E1 -3150,E2 -3150} C_VEL
LIN {X 0,Y 552.174,Z 281.698,A -85,B 0,C 180,E1 -3152.919,E2 -3152.919} C_VEL
LIN {X 0,Y 552.168,Z 281.701,A -85,B 0,C 180,E1 -3155.845,E2 -3155.845} C_VEL
LIN {X 0,Y 552.123,Z 281.708,A -85,B 0,C 180,E1 -3158.787,E2 -3158.787} C_VEL
LIN {X 0,Y 552.074,Z 281.711,A -85,B 0,C 180,E1 -3161.753,E2 -3161.753} C_VEL
LIN {X 0,Y 552.085,Z 281.718,A -85,B 0,C 180,E1 -3164.651,E2 -3164.651} C_VEL
LIN {X 0,Y 552.097,Z 281.708,A -85,B 0,C 180,E1 -3167.305,E2 -3167.305} C_VEL
LIN {X 0,Y 552.095,Z 281.709,A -85,B 0,C 180,E1 -3170.103,E2 -3170.103} C_VEL
LIN {X 0,Y 552.05,Z 281.719,A -85,B 0,C 180,E1 -3172.453,E2 -3172.453} C_VEL
LIN {X 0,Y 552.06,Z 281.717,A -85,B 0,C 180,E1 -3175.328,E2 -3175.328} C_VEL
LIN {X 0,Y 552.103,Z 281.805,A -85,B 0,C 180,E1 -3177.686,E2 -3177.686} C_VEL
LIN {X 0,Y 552.469,Z 286.751,A -85,B 0,C 180,E1 -3178.626,E2 -3178.626} C_VEL
LIN {X 0,Y 552.269,Z 301.885,A -85,B 0,C 180,E1 -3181.45,E2 -3181.45} C_VEL
LIN {X 0,Y 552.206,Z 308.716,A -85,B 0,C 180,E1 -3182.695,E2 -3182.695} C_VEL
LIN {X 0,Y 553.375,Z 315.406,A -85,B 0,C 180,E1 -3182.814,E2 -3182.814} C_VEL
LIN {X 0,Y 553.134,Z 415.943,A -85,B 0,C 180,E1 -3184.146,E2 -3184.146} C_VEL
LIN {X 0,Y 552.935,Z 429.372,A -85,B 0,C 180,E1 -3184.49,E2 -3184.49} C_VEL
LIN {X 0,Y 552.825,Z 440.332,A -85,B 0,C 180,E1 -3184.896,E2 -3184.896} C_VEL
LIN {X 0,Y 552.641,Z 450.591,A -85,B 0,C 180,E1 -3185.387,E2 -3185.387} C_VEL
LIN {X 0,Y 552.485,Z 459.686,A -85,B 0,C 180,E1 -3185.926,E2 -3185.926} C_VEL
LIN {X 0,Y 552.388,Z 467.653,A -85,B 0,C 180,E1 -3186.489,E2 -3186.489} C_VEL
LIN {X 0,Y 552.203,Z 477.25,A -85,B 0,C 180,E1 -3187.311,E2 -3187.311} C_VEL
LIN {X 0,Y 552.113,Z 484.237,A -85,B 0,C 180,E1 -3188.018,E2 -3188.018} C_VEL
LIN {X 0,Y 551.99,Z 490.992,A -85,B 0,C 180,E1 -3188.819,E2 -3188.819} C_VEL
LIN {X 0,Y 551.881,Z 498.211,A -85,B 0,C 180,E1 -3189.856,E2 -3189.856} C_VEL
LIN {X 0,Y 551.796,Z 504.119,A -85,B 0,C 180,E1 -3190.895,E2 -3190.895} C_VEL
LIN {X 0,Y 551.774,Z 508.847,A -85,B 0,C 180,E1 -3191.923,E2 -3191.923} C_VEL
LIN {X 0,Y 551.71,Z 512.582,A -85,B 0,C 180,E1 -3192.948,E2 -3192.948} C_VEL
LIN {X 0,Y 551.708,Z 515.404,A -85,B 0,C 180,E1 -3193.968,E2 -3193.968} C_VEL
LIN {X 0,Y 551.678,Z 517.421,A -85,B 0,C 180,E1 -3195.006,E2 -3195.006} C_VEL
LIN {X 0,Y 551.673,Z 518.84,A -85,B 0,C 180,E1 -3196.565,E2 -3196.565} C_VEL
LIN {X 0,Y 551.66,Z 518.792,A -85,B 0,C 180,E1 -3197.638,E2 -3197.638} C_VEL
LIN {X 0,Y 551.67,Z 517.863,A -85,B 0,C 180,E1 -3198.732,E2 -3198.732} C_VEL
LIN {X 0,Y 551.653,Z 515.971,A -85,B 0,C 180,E1 -3199.853,E2 -3199.853} C_VEL
LIN {X 0,Y 551.678,Z 514.686,A -85,B 0,C 180,E1 -3200.434,E2 -3200.434} C_VEL
LIN {X 0,Y 551.748,Z 510.312,A -85,B 0,C 180,E1 -3201.798,E2 -3201.798} C_VEL
LIN {X 0,Y 551.782,Z 506.228,A -85,B 0,C 180,E1 -3202.77,E2 -3202.77} C_VEL
LIN {X 0,Y 551.854,Z 501.151,A -85,B 0,C 180,E1 -3203.749,E2 -3203.749} C_VEL
LIN {X 0,Y 551.927,Z 494.321,A -85,B 0,C 180,E1 -3204.815,E2 -3204.815} C_VEL
LIN {X 0,Y 552.051,Z 487.616,A -85,B 0,C 180,E1 -3205.683,E2 -3205.683} C_VEL
LIN {X 0,Y 552.165,Z 480.24,A -85,B 0,C 180,E1 -3206.49,E2 -3206.49} C_VEL
LIN {X 0,Y 552.317,Z 472.698,A -85,B 0,C 180,E1 -3207.19,E2 -3207.19} C_VEL
LIN {X 0,Y 552.396,Z 463.559,A -85,B 0,C 180,E1 -3207.902,E2 -3207.902} C_VEL
LIN {X 0,Y 552.604,Z 453.892,A -85,B 0,C 180,E1 -3208.52,E2 -3208.52} C_VEL
LIN {X 0,Y 552.746,Z 443.419,A -85,B 0,C 180,E1 -3209.059,E2 -3209.059} C_VEL
LIN {X 0,Y 552.909,Z 434.084,A -85,B 0,C 180,E1 -3209.44,E2 -3209.44} C_VEL
LIN {X 0,Y 552.978,Z 423.594,A -85,B 0,C 180,E1 -3209.765,E2 -3209.765} C_VEL
LIN {X 0,Y 553.107,Z 411.531,A -85,B 0,C 180,E1 -3210.017,E2 -3210.017} C_VEL
LIN {X 0,Y 553.285,Z 315.018,A -85,B 0,C 180,E1 -3211.283,E2 -3211.283} C_VEL
LIN {X 0,Y 552.145,Z 308.456,A -85,B 0,C 180,E1 -3211.411,E2 -3211.411} C_VEL
LIN {X 0,Y 552.245,Z 298.029,A -85,B 0,C 180,E1 -3213.259,E2 -3213.259} C_VEL
LIN {X 0,Y 552.296,Z 288.55,A -85,B 0,C 180,E1 -3214.89,E2 -3214.89} C_VEL
LIN {X 0,Y 552.221,Z 281.698,A -85,B 0,C 180,E1 -3216,E2 -3216} C_VEL
LIN {X 0,Y 552.121,Z 281.714,A -85,B 0,C 180,E1 -3219.12,E2 -3219.12} C_VEL
LIN {X 0,Y 552.123,Z 281.715,A -85,B 0,C 180,E1 -3221.444,E2 -3221.444} C_VEL
LIN {X 0,Y 552.117,Z 281.712,A -85,B 0,C 180,E1 -3223.737,E2 -3223.737} C_VEL
LIN {X 0,Y 552.137,Z 281.706,A -85,B 0,C 180,E1 -3226.004,E2 -3226.004} C_VEL
LIN {X 0,Y 552.163,Z 281.701,A -85,B 0,C 180,E1 -3228.993,E2 -3228.993} C_VEL
LIN {X 0,Y 552.151,Z 281.707,A -85,B 0,C 180,E1 -3231.951,E2 -3231.951} C_VEL
LIN {X 0,Y 552.227,Z 281.692,A -85,B 0,C 180,E1 -3234.889,E2 -3234.889} C_VEL
LIN {X 0,Y 552.223,Z 281.702,A -85,B 0,C 180,E1 -3237.812,E2 -3237.812} C_VEL
LIN {X 0,Y 552.241,Z 281.689,A -85,B 0,C 180,E1 -3240.729,E2 -3240.729} C_VEL
LIN {X 0,Y 552.203,Z 281.694,A -85,B 0,C 180,E1 -3242.918,E2 -3242.918} C_VEL
LIN {X 0,Y 552.192,Z 281.701,A -85,B 0,C 180,E1 -3245.844,E2 -3245.844} C_VEL
LIN {X 0,Y 552.154,Z 281.702,A -85,B 0,C 180,E1 -3248.786,E2 -3248.786} C_VEL
LIN {X 0,Y 552.164,Z 281.701,A -85,B 0,C 180,E1 -3251.75,E2 -3251.75} C_VEL
LIN {X 0,Y 552.138,Z 281.707,A -85,B 0,C 180,E1 -3254.748,E2 -3254.748} C_VEL
LIN {X 0,Y 552.101,Z 281.706,A -85,B 0,C 180,E1 -3257.789,E2 -3257.789} C_VEL
LIN {X 0,Y 552.128,Z 281.706,A -85,B 0,C 180,E1 -3260.101,E2 -3260.101} C_VEL
LIN {X 0,Y 552.093,Z 281.714,A -85,B 0,C 180,E1 -3262.451,E2 -3262.451} C_VEL
LIN {X 0,Y 552.157,Z 281.701,A -85,B 0,C 180,E1 -3265.35,E2 -3265.35} C_VEL
LIN {X 0,Y 552.107,Z 281.705,A -85,B 0,C 180,E1 -3268.098,E2 -3268.098} C_VEL
LIN {X 0,Y 552.104,Z 281.712,A -85,B 0,C 180,E1 -3270.609,E2 -3270.609} C_VEL
LIN {X 0,Y 552.107,Z 281.713,A -85,B 0,C 180,E1 -3273.186,E2 -3273.186} C_VEL
LIN {X 0,Y 552.087,Z 281.709,A -85,B 0,C 180,E1 -3275.844,E2 -3275.844} C_VEL
LIN {X 0,Y 552.119,Z 281.706,A -85,B 0,C 180,E1 -3278.589,E2 -3278.589} C_VEL
LIN {X 0,Y 552.123,Z 281.712,A -85,B 0,C 180,E1 -3281.446,E2 -3281.446} C_VEL
LIN {X 0,Y 552.09,Z 281.709,A -85,B 0,C 180,E1 -3284.531,E2 -3284.531} C_VEL
LIN {X 0,Y 552.132,Z 281.712,A -85,B 0,C 180,E1 -3287.585,E2 -3287.585} C_VEL
LIN {X 0,Y 552.131,Z 281.704,A -85,B 0,C 180,E1 -3290.473,E2 -3290.473} C_VEL
LIN {X 0,Y 552.109,Z 281.712,A -85,B 0,C 180,E1 -3293.317,E2 -3293.317} C_VEL
LIN {X 0,Y 552.128,Z 281.713,A -85,B 0,C 180,E1 -3295.939,E2 -3295.939} C_VEL
LIN {X 0,Y 552.122,Z 281.706,A -85,B 0,C 180,E1 -3298.541,E2 -3298.541} C_VEL
LIN {X 0,Y 552.127,Z 281.708,A -85,B 0,C 180,E1 -3301.438,E2 -3301.438} C_VEL
LIN {X 0,Y 552.131,Z 281.711,A -85,B 0,C 180,E1 -3304.356,E2 -3304.356} C_VEL
LIN {X 0,Y 552.134,Z 281.82,A -85,B 0,C 180,E1 -3306.199,E2 -3306.199} C_VEL
LIN {X 0,Y 553.112,Z 288.358,A -85,B 0,C 180,E1 -3307.198,E2 -3307.198} C_VEL
LIN {X 0,Y 552.828,Z 308.738,A -85,B 0,C 180,E1 -3310.178,E2 -3310.178} C_VEL
LIN {X 0,Y 552.58,Z 328.25,A -85,B 0,C 180,E1 -3312.99,E2 -3312.99} C_VEL
LIN {X 0,Y 552.374,Z 346.704,A -85,B 0,C 180,E1 -3315.625,E2 -3315.625} C_VEL
LIN {X 0,Y 553.416,Z 354.758,A -85,B 0,C 180,E1 -3315.762,E2 -3315.762} C_VEL
LIN {X 0,Y 553.101,Z 454.929,A -85,B 0,C 180,E1 -3317.082,E2 -3317.082} C_VEL
LIN {X 0,Y 552.996,Z 468.205,A -85,B 0,C 180,E1 -3317.406,E2 -3317.406} C_VEL
LIN {X 0,Y 552.84,Z 480.36,A -85,B 0,C 180,E1 -3317.845,E2 -3317.845} C_VEL
LIN {X 0,Y 552.695,Z 492.618,A -85,B 0,C 180,E1 -3318.447,E2 -3318.447} C_VEL
LIN {X 0,Y 552.5,Z 504.189,A -85,B 0,C 180,E1 -3319.185,E2 -3319.185} C_VEL
LIN {X 0,Y 552.295,Z 514.601,A -85,B 0,C 180,E1 -3320.015,E2 -3320.015} C_VEL
LIN {X 0,Y 552.126,Z 523.106,A -85,B 0,C 180,E1 -3320.844,E2 -3320.844} C_VEL
LIN {X 0,Y 552.009,Z 530.958,A -85,B 0,C 180,E1 -3321.765,E2 -3321.765} C_VEL
LIN {X 0,Y 551.89,Z 538.619,A -85,B 0,C 180,E1 -3322.867,E2 -3322.867} C_VEL
LIN {X 0,Y 551.868,Z 545.678,A -85,B 0,C 180,E1 -3324.152,E2 -3324.152} C_VEL
LIN {X 0,Y 551.725,Z 550.371,A -85,B 0,C 180,E1 -3325.25,E2 -3325.25} C_VEL
LIN {X 0,Y 551.75,Z 553.957,A -85,B 0,C 180,E1 -3326.348,E2 -3326.348} C_VEL
LIN {X 0,Y 551.723,Z 555.806,A -85,B 0,C 180,E1 -3327.079,E2 -3327.079} C_VEL
LIN {X 0,Y 551.644,Z 558.183,A -85,B 0,C 180,E1 -3328.54,E2 -3328.54} C_VEL
LIN {X 0,Y 551.64,Z 559,A -85,B 0,C 180,E1 -3330,E2 -3330} C_VEL
LIN {X 0,Y 551.645,Z 558.185,A -85,B 0,C 180,E1 -3331.46,E2 -3331.46} C_VEL
LIN {X 0,Y 551.723,Z 555.811,A -85,B 0,C 180,E1 -3332.92,E2 -3332.92} C_VEL
LIN {X 0,Y 551.763,Z 552.897,A -85,B 0,C 180,E1 -3334.017,E2 -3334.017} C_VEL
LIN {X 0,Y 551.723,Z 548.95,A -85,B 0,C 180,E1 -3335.115,E2 -3335.115} C_VEL
LIN {X 0,Y 551.814,Z 543.127,A -85,B 0,C 180,E1 -3336.353,E2 -3336.353} C_VEL
LIN {X 0,Y 551.926,Z 536.239,A -85,B 0,C 180,E1 -3337.499,E2 -3337.499} C_VEL
LIN {X 0,Y 552.063,Z 527.996,A -85,B 0,C 180,E1 -3338.602,E2 -3338.602} C_VEL
LIN {X 0,Y 552.222,Z 519.545,A -85,B 0,C 180,E1 -3339.523,E2 -3339.523} C_VEL
LIN {X 0,Y 552.406,Z 509.098,A -85,B 0,C 180,E1 -3340.445,E2 -3340.445} C_VEL
LIN {X 0,Y 552.609,Z 498.198,A -85,B 0,C 180,E1 -3341.219,E2 -3341.219} C_VEL
LIN {X 0,Y 552.749,Z 487.414,A -85,B 0,C 180,E1 -3341.83,E2 -3341.83} C_VEL
LIN {X 0,Y 552.883,Z 475.778,A -85,B 0,C 180,E1 -3342.34,E2 -3342.34} C_VEL
LIN {X 0,Y 553.005,Z 462.365,A -85,B 0,C 180,E1 -3342.756,E2 -3342.756} C_VEL
LIN {X 0,Y 553.182,Z 449.121,A -85,B 0,C 180,E1 -3343.009,E2 -3343.009} C_VEL
LIN {X 0,Y 553.255,Z 352.366,A -85,B 0,C 180,E1 -3344.273,E2 -3344.273} C_VEL
LIN {X 0,Y 552.381,Z 346.659,A -85,B 0,C 180,E1 -3344.381,E2 -3344.381} C_VEL
LIN {X 0,Y 552.632,Z 325.188,A -85,B 0,C 180,E1 -3347.484,E2 -3347.484} C_VEL
LIN {X 0,Y 552.93,Z 306.174,A -85,B 0,C 180,E1 -3350.264,E2 -3350.264} C_VEL
LIN {X 0,Y 553.226,Z 287.807,A -85,B 0,C 180,E1 -3352.994,E2 -3352.994} C_VEL
LIN {X 0,Y 552.144,Z 281.712,A -85,B 0,C 180,E1 -3353.977,E2 -3353.977} C_VEL
LIN {X 0,Y 552.118,Z 281.71,A -85,B 0,C 180,E1 -3356.456,E2 -3356.456} C_VEL
LIN {X 0,Y 552.109,Z 281.706,A -85,B 0,C 180,E1 -3358.928,E2 -3358.928} C_VEL
LIN {X 0,Y 552.11,Z 281.707,A -85,B 0,C 180,E1 -3361.475,E2 -3361.475} C_VEL
LIN {X 0,Y 552.131,Z 281.713,A -85,B 0,C 180,E1 -3364.17,E2 -3364.17} C_VEL
LIN {X 0,Y 552.103,Z 281.709,A -85,B 0,C 180,E1 -3366.746,E2 -3366.746} C_VEL
LIN {X 0,Y 552.127,Z 281.703,A -85,B 0,C 180,E1 -3369.527,E2 -3369.527} C_VEL
LIN {X 0,Y 552.128,Z 281.714,A -85,B 0,C 180,E1 -3372.425,E2 -3372.425} C_VEL
LIN {X 0,Y 552.094,Z 281.707,A -85,B 0,C 180,E1 -3375.562,E2 -3375.562} C_VEL
LIN {X 0,Y 552.137,Z 281.711,A -85,B 0,C 180,E1 -3378.675,E2 -3378.675} C_VEL
LIN {X 0,Y 552.116,Z 281.705,A -85,B 0,C 180,E1 -3381.411,E2 -3381.411} C_VEL
LIN {X 0,Y 552.098,Z 281.709,A -85,B 0,C 180,E1 -3384.157,E2 -3384.157} C_VEL
LIN {X 0,Y 552.118,Z 281.715,A -85,B 0,C 180,E1 -3386.814,E2 -3386.814} C_VEL
LIN {X 0,Y 552.103,Z 281.709,A -85,B 0,C 180,E1 -3389.391,E2 -3389.391} C_VEL
LIN {X 0,Y 552.114,Z 281.705,A -85,B 0,C 180,E1 -3391.902,E2 -3391.902} C_VEL
LIN {X 0,Y 552.15,Z 281.704,A -85,B 0,C 180,E1 -3394.649,E2 -3394.649} C_VEL
LIN {X 0,Y 552.09,Z 281.711,A -85,B 0,C 180,E1 -3397.549,E2 -3397.549} C_VEL
LIN {X 0,Y 552.143,Z 281.702,A -85,B 0,C 180,E1 -3400.373,E2 -3400.373} C_VEL
LIN {X 0,Y 552.149,Z 281.706,A -85,B 0,C 180,E1 -3402.977,E2 -3402.977} C_VEL
LIN {X 0,Y 552.13,Z 281.704,A -85,B 0,C 180,E1 -3406.004,E2 -3406.004} C_VEL
LIN {X 0,Y 552.156,Z 281.703,A -85,B 0,C 180,E1 -3408.993,E2 -3408.993} C_VEL
LIN {X 0,Y 552.155,Z 281.703,A -85,B 0,C 180,E1 -3411.952,E2 -3411.952} C_VEL
LIN {X 0,Y 552.224,Z 281.692,A -85,B 0,C 180,E1 -3414.889,E2 -3414.889} C_VEL
LIN {X 0,Y 552.213,Z 281.7,A -85,B 0,C 180,E1 -3417.812,E2 -3417.812} C_VEL
LIN {X 0,Y 552.234,Z 281.69,A -85,B 0,C 180,E1 -3420.729,E2 -3420.729} C_VEL
LIN {X 0,Y 552.198,Z 281.694,A -85,B 0,C 180,E1 -3422.918,E2 -3422.918} C_VEL
LIN {X 0,Y 552.191,Z 281.705,A -85,B 0,C 180,E1 -3425.844,E2 -3425.844} C_VEL
LIN {X 0,Y 552.151,Z 281.7,A -85,B 0,C 180,E1 -3428.786,E2 -3428.786} C_VEL
LIN {X 0,Y 552.157,Z 281.705,A -85,B 0,C 180,E1 -3431.751,E2 -3431.751} C_VEL
LIN {X 0,Y 552.123,Z 281.705,A -85,B 0,C 180,E1 -3434.749,E2 -3434.749} C_VEL
LIN {X 0,Y 552.093,Z 281.711,A -85,B 0,C 180,E1 -3437.789,E2 -3437.789} C_VEL
LIN {X 0,Y 552.121,Z 281.712,A -85,B 0,C 180,E1 -3440.102,E2 -3440.102} C_VEL
LIN {X 0,Y 552.086,Z 281.717,A -85,B 0,C 180,E1 -3442.452,E2 -3442.452} C_VEL
LIN {X 0,Y 552.133,Z 281.702,A -85,B 0,C 180,E1 -3445.347,E2 -3445.347} C_VEL
LIN {X 0,Y 552.073,Z 281.714,A -85,B 0,C 180,E1 -3448.101,E2 -3448.101} C_VEL
LIN {X 0,Y 552.097,Z 281.717,A -85,B 0,C 180,E1 -3450.61,E2 -3450.61} C_VEL
LIN {X 0,Y 552.108,Z 281.708,A -85,B 0,C 180,E1 -3453.187,E2 -3453.187} C_VEL
LIN {X 0,Y 552.104,Z 281.706,A -85,B 0,C 180,E1 -3453.775,E2 -3453.775} C_VEL
LIN {X 0,Y 551.47,Z 281.792,A -85,B 0,C 180,E1 -3454.383,E2 -3454.383} C_VEL
LIN {X 0,Y 548.651,Z 282.148,A -85,B 0,C 180,E1 -3455.372,E2 -3455.372} C_VEL
LIN {X 0,Y 546.231,Z 282.451,A -85,B 0,C 180,E1 -3456.167,E2 -3456.167} C_VEL
LIN {X 0,Y 545.162,Z 282.581,A -85,B 0,C 180,E1 -3456.781,E2 -3456.781} C_VEL
LIN {X 0,Y 545.059,Z 282.59,A -85,B 0,C 180,E1 -3456.989,E2 -3456.989} C_VEL
LIN {X 0,Y 545.061,Z 282.585,A -85,B 0,C 180,E1 -3460.144,E2 -3460.144} C_VEL
LIN {X 0,Y 545.036,Z 282.594,A -85,B 0,C 180,E1 -3462.695,E2 -3462.695} C_VEL
LIN {X 0,Y 545.027,Z 282.594,A -85,B 0,C 180,E1 -3465.171,E2 -3465.171} C_VEL
LIN {X 0,Y 545.05,Z 282.585,A -85,B 0,C 180,E1 -3467.895,E2 -3467.895} C_VEL
LIN {X 0,Y 545.075,Z 282.587,A -85,B 0,C 180,E1 -3470.819,E2 -3470.819} C_VEL
LIN {X 0,Y 545.034,Z 282.59,A -85,B 0,C 180,E1 -3473.62,E2 -3473.62} C_VEL
LIN {X 0,Y 545.048,Z 282.585,A -85,B 0,C 180,E1 -3476.328,E2 -3476.328} C_VEL
LIN {X 0,Y 545.053,Z 282.589,A -85,B 0,C 180,E1 -3478.952,E2 -3478.952} C_VEL
LIN {X 0,Y 545.042,Z 282.594,A -85,B 0,C 180,E1 -3481.505,E2 -3481.505} C_VEL
LIN {X 0,Y 545.03,Z 282.587,A -85,B 0,C 180,E1 -3484.507,E2 -3484.507} C_VEL
LIN {X 0,Y 545.035,Z 282.592,A -85,B 0,C 180,E1 -3487.243,E2 -3487.243} C_VEL
LIN {X 0,Y 545.094,Z 282.581,A -85,B 0,C 180,E1 -3490.256,E2 -3490.256} C_VEL
LIN {X 0,Y 545.053,Z 282.584,A -85,B 0,C 180,E1 -3492.749,E2 -3492.749} C_VEL
LIN {X 0,Y 545.091,Z 282.59,A -85,B 0,C 180,E1 -3495.82,E2 -3495.82} C_VEL
LIN {X 0,Y 545.074,Z 282.582,A -85,B 0,C 180,E1 -3498.849,E2 -3498.849} C_VEL
LIN {X 0,Y 545.068,Z 282.591,A -85,B 0,C 180,E1 -3501.847,E2 -3501.847} C_VEL
LIN {X 0,Y 545.162,Z 282.571,A -85,B 0,C 180,E1 -3504.823,E2 -3504.823} C_VEL
LIN {X 0,Y 545.192,Z 282.572,A -85,B 0,C 180,E1 -3507.784,E2 -3507.784} C_VEL
LIN {X 0,Y 545.194,Z 282.574,A -85,B 0,C 180,E1 -3510,E2 -3510} C_VEL
LIN {X 0,Y 545.142,Z 282.574,A -85,B 0,C 180,E1 -3512.956,E2 -3512.956} C_VEL
LIN {X 0,Y 545.123,Z 282.579,A -85,B 0,C 180,E1 -3515.92,E2 -3515.92} C_VEL
LIN {X 0,Y 545.066,Z 282.586,A -85,B 0,C 180,E1 -3518.901,E2 -3518.901} C_VEL
LIN {X 0,Y 545.05,Z 282.587,A -85,B 0,C 180,E1 -3521.906,E2 -3521.906} C_VEL
LIN {X 0,Y 545.04,Z 282.59,A -85,B 0,C 180,E1 -3524.945,E2 -3524.945} C_VEL
LIN {X 0,Y 545.048,Z 282.587,A -85,B 0,C 180,E1 -3528.027,E2 -3528.027} C_VEL
LIN {X 0,Y 545.034,Z 282.591,A -85,B 0,C 180,E1 -3530.375,E2 -3530.375} C_VEL
LIN {X 0,Y 545.004,Z 282.601,A -85,B 0,C 180,E1 -3532.76,E2 -3532.76} C_VEL
LIN {X 0,Y 545.004,Z 282.595,A -85,B 0,C 180,E1 -3535.487,E2 -3535.487} C_VEL
LIN {X 0,Y 545.063,Z 282.619,A -85,B 0,C 180,E1 -3537.578,E2 -3537.578} C_VEL
LIN {X 0,Y 545.463,Z 287.26,A -85,B 0,C 180,E1 -3538.472,E2 -3538.472} C_VEL
LIN {X 0,Y 545.267,Z 302.668,A -85,B 0,C 180,E1 -3541.367,E2 -3541.367} C_VEL
LIN {X 0,Y 545.194,Z 308.758,A -85,B 0,C 180,E1 -3542.506,E2 -3542.506} C_VEL
LIN {X 0,Y 546.479,Z 316.096,A -85,B 0,C 180,E1 -3542.639,E2 -3542.639} C_VEL
LIN {X 0,Y 546.227,Z 415.864,A -85,B 0,C 180,E1 -3543.979,E2 -3543.979} C_VEL
LIN {X 0,Y 546.015,Z 429.467,A -85,B 0,C 180,E1 -3544.328,E2 -3544.328} C_VEL
LIN {X 0,Y 545.889,Z 440.51,A -85,B 0,C 180,E1 -3544.742,E2 -3544.742} C_VEL
LIN {X 0,Y 545.702,Z 450.617,A -85,B 0,C 180,E1 -3545.232,E2 -3545.232} C_VEL
LIN {X 0,Y 545.519,Z 459.202,A -85,B 0,C 180,E1 -3545.743,E2 -3545.743} C_VEL
LIN {X 0,Y 545.363,Z 469.032,A -85,B 0,C 180,E1 -3546.461,E2 -3546.461} C_VEL
LIN {X 0,Y 545.189,Z 477.371,A -85,B 0,C 180,E1 -3547.193,E2 -3547.193} C_VEL
LIN {X 0,Y 545.062,Z 484.667,A -85,B 0,C 180,E1 -3547.95,E2 -3547.95} C_VEL
LIN {X 0,Y 544.948,Z 491.027,A -85,B 0,C 180,E1 -3548.718,E2 -3548.718} C_VEL
LIN {X 0,Y 544.828,Z 497.844,A -85,B 0,C 180,E1 -3549.703,E2 -3549.703} C_VEL
LIN {X 0,Y 544.725,Z 503.858,A -85,B 0,C 180,E1 -3550.763,E2 -3550.763} C_VEL
LIN {X 0,Y 544.681,Z 508.704,A -85,B 0,C 180,E1 -3551.821,E2 -3551.821} C_VEL
LIN {X 0,Y 544.659,Z 511.841,A -85,B 0,C 180,E1 -3552.65,E2 -3552.65} C_VEL
LIN {X 0,Y 544.605,Z 514.962,A -85,B 0,C 180,E1 -3553.724,E2 -3553.724} C_VEL
LIN {X 0,Y 544.575,Z 517.139,A -85,B 0,C 180,E1 -3554.781,E2 -3554.781} C_VEL
LIN {X 0,Y 544.564,Z 518.449,A -85,B 0,C 180,E1 -3555.82,E2 -3555.82} C_VEL
LIN {X 0,Y 544.554,Z 518.947,A -85,B 0,C 180,E1 -3556.841,E2 -3556.841} C_VEL
LIN {X 0,Y 544.561,Z 518.699,A -85,B 0,C 180,E1 -3557.847,E2 -3557.847} C_VEL
LIN {X 0,Y 544.565,Z 517.75,A -85,B 0,C 180,E1 -3558.837,E2 -3558.837} C_VEL
LIN {X 0,Y 544.597,Z 515.107,A -85,B 0,C 180,E1 -3560.298,E2 -3560.298} C_VEL
LIN {X 0,Y 544.655,Z 510.812,A -85,B 0,C 180,E1 -3561.729,E2 -3561.729} C_VEL
LIN {X 0,Y 544.707,Z 505.84,A -85,B 0,C 180,E1 -3562.922,E2 -3562.922} C_VEL
LIN {X 0,Y 544.78,Z 501.34,A -85,B 0,C 180,E1 -3563.803,E2 -3563.803} C_VEL
LIN {X 0,Y 544.852,Z 495.548,A -85,B 0,C 180,E1 -3564.744,E2 -3564.744} C_VEL
LIN {X 0,Y 544.995,Z 487.983,A -85,B 0,C 180,E1 -3565.752,E2 -3565.752} C_VEL
LIN {X 0,Y 545.138,Z 479.859,A -85,B 0,C 180,E1 -3566.653,E2 -3566.653} C_VEL
LIN {X 0,Y 545.31,Z 471.253,A -85,B 0,C 180,E1 -3567.447,E2 -3567.447} C_VEL
LIN {X 0,Y 545.437,Z 462.668,A -85,B 0,C 180,E1 -3568.11,E2 -3568.11} C_VEL
LIN {X 0,Y 545.635,Z 454.067,A -85,B 0,C 180,E1 -3568.664,E2 -3568.664} C_VEL
LIN {X 0,Y 545.785,Z 444.624,A -85,B 0,C 180,E1 -3569.165,E2 -3569.165} C_VEL
LIN {X 0,Y 545.968,Z 434.363,A -85,B 0,C 180,E1 -3569.594,E2 -3569.594} C_VEL
LIN {X 0,Y 546.047,Z 423.387,A -85,B 0,C 180,E1 -3569.937,E2 -3569.937} C_VEL
LIN {X 0,Y 546.193,Z 411.453,A -85,B 0,C 180,E1 -3570.185,E2 -3570.185} C_VEL
LIN {X 0,Y 546.446,Z 315.995,A -85,B 0,C 180,E1 -3571.452,E2 -3571.452} C_VEL
LIN {X 0,Y 545.154,Z 308.651,A -85,B 0,C 180,E1 -3571.589,E2 -3571.589} C_VEL
LIN {X 0,Y 545.196,Z 297.069,A -85,B 0,C 180,E1 -3573.593,E2 -3573.593} C_VEL
LIN {X 0,Y 545.261,Z 287.313,A -85,B 0,C 180,E1 -3575.234,E2 -3575.234} C_VEL
LIN {X 0,Y 545.183,Z 282.575,A -85,B 0,C 180,E1 -3576.013,E2 -3576.013} C_VEL
LIN {X 0,Y 545.095,Z 282.586,A -85,B 0,C 180,E1 -3579.628,E2 -3579.628} C_VEL
LIN {X 0,Y 545.08,Z 282.585,A -85,B 0,C 180,E1 -3582.749,E2 -3582.749} C_VEL
LIN {X 0,Y 545.096,Z 282.586,A -85,B 0,C 180,E1 -3585.82,E2 -3585.82} C_VEL
LIN {X 0,Y 545.119,Z 282.578,A -85,B 0,C 180,E1 -3588.849,E2 -3588.849} C_VEL
LIN {X 0,Y 545.122,Z 282.584,A -85,B 0,C 180,E1 -3591.847,E2 -3591.847} C_VEL
LIN {X 0,Y 545.203,Z 282.567,A -85,B 0,C 180,E1 -3594.823,E2 -3594.823} C_VEL
LIN {X 0,Y 545.195,Z 282.577,A -85,B 0,C 180,E1 -3597.783,E2 -3597.783} C_VEL
LIN {X 0,Y 545.211,Z 282.565,A -85,B 0,C 180,E1 -3600.738,E2 -3600.738} C_VEL
LIN {X 0,Y 545.17,Z 282.57,A -85,B 0,C 180,E1 -3602.956,E2 -3602.956} C_VEL
LIN {X 0,Y 545.162,Z 282.578,A -85,B 0,C 180,E1 -3605.919,E2 -3605.919} C_VEL
LIN {X 0,Y 545.112,Z 282.578,A -85,B 0,C 180,E1 -3608.9,E2 -3608.9} C_VEL
LIN {X 0,Y 545.136,Z 282.578,A -85,B 0,C 180,E1 -3611.904,E2 -3611.904} C_VEL
LIN {X 0,Y 545.087,Z 282.583,A -85,B 0,C 180,E1 -3614.943,E2 -3614.943} C_VEL
LIN {X 0,Y 545.073,Z 282.584,A -85,B 0,C 180,E1 -3618.026,E2 -3618.026} C_VEL
LIN {X 0,Y 545.094,Z 282.586,A -85,B 0,C 180,E1 -3620.372,E2 -3620.372} C_VEL
LIN {X 0,Y 545.08,Z 282.581,A -85,B 0,C 180,E1 -3623.559,E2 -3623.559} C_VEL
LIN {X 0,Y 545.081,Z 282.581,A -85,B 0,C 180,E1 -3626,E2 -3626} C_VEL
LIN {X 0,Y 545.091,Z 282.587,A -85,B 0,C 180,E1 -3628.748,E2 -3628.748} C_VEL
LIN {X 0,Y 545.059,Z 282.584,A -85,B 0,C 180,E1 -3631.679,E2 -3631.679} C_VEL
LIN {X 0,Y 545.06,Z 282.587,A -85,B 0,C 180,E1 -3634.565,E2 -3634.565} C_VEL
LIN {X 0,Y 545.038,Z 282.594,A -85,B 0,C 180,E1 -3637.304,E2 -3637.304} C_VEL
LIN {X 0,Y 545.067,Z 282.583,A -85,B 0,C 180,E1 -3640.143,E2 -3640.143} C_VEL
LIN {X 0,Y 545.08,Z 282.589,A -85,B 0,C 180,E1 -3643.107,E2 -3643.107} C_VEL
LIN {X 0,Y 545.051,Z 282.586,A -85,B 0,C 180,E1 -3646.226,E2 -3646.226} C_VEL
LIN {X 0,Y 545.083,Z 282.583,A -85,B 0,C 180,E1 -3648.885,E2 -3648.885} C_VEL
LIN {X 0,Y 545.054,Z 282.594,A -85,B 0,C 180,E1 -3651.763,E2 -3651.763} C_VEL
LIN {X 0,Y 545.038,Z 282.589,A -85,B 0,C 180,E1 -3654.531,E2 -3654.531} C_VEL
LIN {X 0,Y 545.069,Z 282.587,A -85,B 0,C 180,E1 -3657.211,E2 -3657.211} C_VEL
LIN {X 0,Y 545.066,Z 282.593,A -85,B 0,C 180,E1 -3659.81,E2 -3659.81} C_VEL
LIN {X 0,Y 545.078,Z 282.589,A -85,B 0,C 180,E1 -3662.343,E2 -3662.343} C_VEL
LIN {X 0,Y 545.109,Z 282.582,A -85,B 0,C 180,E1 -3664.82,E2 -3664.82} C_VEL
LIN {X 0,Y 545.109,Z 282.637,A -85,B 0,C 180,E1 -3666.066,E2 -3666.066} C_VEL
LIN {X 0,Y 546.151,Z 289.312,A -85,B 0,C 180,E1 -3667.091,E2 -3667.091} C_VEL
LIN {X 0,Y 545.872,Z 308.313,A -85,B 0,C 180,E1 -3669.903,E2 -3669.903} C_VEL
LIN {X 0,Y 545.562,Z 329.212,A -85,B 0,C 180,E1 -3672.958,E2 -3672.958} C_VEL
LIN {X 0,Y 545.349,Z 346.449,A -85,B 0,C 180,E1 -3675.444,E2 -3675.444} C_VEL
LIN {X 0,Y 546.524,Z 354.708,A -85,B 0,C 180,E1 -3675.584,E2 -3675.584} C_VEL
LIN {X 0,Y 546.183,Z 454.667,A -85,B 0,C 180,E1 -3676.915,E2 -3676.915} C_VEL
LIN {X 0,Y 546.06,Z 468.027,A -85,B 0,C 180,E1 -3677.243,E2 -3677.243} C_VEL
LIN {X 0,Y 545.886,Z 480.247,A -85,B 0,C 180,E1 -3677.688,E2 -3677.688} C_VEL
LIN {X 0,Y 545.736,Z 492.575,A -85,B 0,C 180,E1 -3678.297,E2 -3678.297} C_VEL
LIN {X 0,Y 545.522,Z 504.187,A -85,B 0,C 180,E1 -3679.045,E2 -3679.045} C_VEL
LIN {X 0,Y 545.282,Z 514.6,A -85,B 0,C 180,E1 -3679.886,E2 -3679.886} C_VEL
LIN {X 0,Y 545.085,Z 523.11,A -85,B 0,C 180,E1 -3680.725,E2 -3680.725} C_VEL
LIN {X 0,Y 544.972,Z 530.958,A -85,B 0,C 180,E1 -3681.658,E2 -3681.658} C_VEL
LIN {X 0,Y 544.824,Z 538.619,A -85,B 0,C 180,E1 -3682.774,E2 -3682.774} C_VEL
LIN {X 0,Y 544.779,Z 545.677,A -85,B 0,C 180,E1 -3684.076,E2 -3684.076} C_VEL
LIN {X 0,Y 544.628,Z 550.371,A -85,B 0,C 180,E1 -3685.188,E2 -3685.188} C_VEL
LIN {X 0,Y 544.669,Z 553.957,A -85,B 0,C 180,E1 -3686.301,E2 -3686.301} C_VEL
LIN {X 0,Y 544.65,Z 555.806,A -85,B 0,C 180,E1 -3687.041,E2 -3687.041} C_VEL
LIN {X 0,Y 544.545,Z 558.182,A -85,B 0,C 180,E1 -3688.52,E2 -3688.52} C_VEL
LIN {X 0,Y 544.541,Z 559,A -85,B 0,C 180,E1 -3690,E2 -3690} C_VEL
LIN {X 0,Y 544.545,Z 558.184,A -85,B 0,C 180,E1 -3691.479,E2 -3691.479} C_VEL
LIN {X 0,Y 544.65,Z 555.811,A -85,B 0,C 180,E1 -3692.958,E2 -3692.958} C_VEL
LIN {X 0,Y 544.683,Z 552.897,A -85,B 0,C 180,E1 -3694.069,E2 -3694.069} C_VEL
LIN {X 0,Y 544.653,Z 548.95,A -85,B 0,C 180,E1 -3695.182,E2 -3695.182} C_VEL
LIN {X 0,Y 544.729,Z 543.646,A -85,B 0,C 180,E1 -3696.339,E2 -3696.339} C_VEL
LIN {X 0,Y 544.859,Z 536.238,A -85,B 0,C 180,E1 -3697.597,E2 -3697.597} C_VEL
LIN {X 0,Y 545.016,Z 527.996,A -85,B 0,C 180,E1 -3698.714,E2 -3698.714} C_VEL
LIN {X 0,Y 545.201,Z 519.545,A -85,B 0,C 180,E1 -3699.647,E2 -3699.647} C_VEL
LIN {X 0,Y 545.386,Z 509.097,A -85,B 0,C 180,E1 -3700.581,E2 -3700.581} C_VEL
LIN {X 0,Y 545.623,Z 497.385,A -85,B 0,C 180,E1 -3701.417,E2 -3701.417} C_VEL
LIN {X 0,Y 545.823,Z 485.42,A -85,B 0,C 180,E1 -3702.077,E2 -3702.077} C_VEL
LIN {X 0,Y 545.981,Z 473.043,A -85,B 0,C 180,E1 -3702.592,E2 -3702.592} C_VEL
LIN {X 0,Y 546.14,Z 460.34,A -85,B 0,C 180,E1 -3702.967,E2 -3702.967} C_VEL
LIN {X 0,Y 546.26,Z 445.299,A -85,B 0,C 180,E1 -3703.224,E2 -3703.224} C_VEL
LIN {X 0,Y 546.406,Z 353.392,A -85,B 0,C 180,E1 -3704.437,E2 -3704.437} C_VEL
LIN {X 0,Y 545.369,Z 346.531,A -85,B 0,C 180,E1 -3704.559,E2 -3704.559} C_VEL
LIN {X 0,Y 545.711,Z 323.01,A -85,B 0,C 180,E1 -3708.004,E2 -3708.004} C_VEL
LIN {X 0,Y 546.004,Z 304.647,A -85,B 0,C 180,E1 -3710.73,E2 -3710.73} C_VEL
LIN {X 0,Y 546.262,Z 288.932,A -85,B 0,C 180,E1 -3713.103,E2 -3713.103} C_VEL
LIN {X 0,Y 545.084,Z 282.591,A -85,B 0,C 180,E1 -3714.164,E2 -3714.164} C_VEL
LIN {X 0,Y 545.093,Z 282.582,A -85,B 0,C 180,E1 -3717.173,E2 -3717.173} C_VEL
LIN {X 0,Y 545.064,Z 282.585,A -85,B 0,C 180,E1 -3719.338,E2 -3719.338} C_VEL
LIN {X 0,Y 545.054,Z 282.591,A -85,B 0,C 180,E1 -3721.914,E2 -3721.914} C_VEL
LIN {X 0,Y 545.061,Z 282.588,A -85,B 0,C 180,E1 -3724.564,E2 -3724.564} C_VEL
LIN {X 0,Y 545.034,Z 282.587,A -85,B 0,C 180,E1 -3727.303,E2 -3727.303} C_VEL
LIN {X 0,Y 545.063,Z 282.59,A -85,B 0,C 180,E1 -3730.142,E2 -3730.142} C_VEL
LIN {X 0,Y 545.075,Z 282.583,A -85,B 0,C 180,E1 -3733.106,E2 -3733.106} C_VEL
LIN {X 0,Y 545.059,Z 282.589,A -85,B 0,C 180,E1 -3736.224,E2 -3736.224} C_VEL
LIN {X 0,Y 545.094,Z 282.585,A -85,B 0,C 180,E1 -3738.886,E2 -3738.886} C_VEL
LIN {X 0,Y 545.05,Z 282.585,A -85,B 0,C 180,E1 -3741.762,E2 -3741.762} C_VEL
LIN {X 0,Y 545.048,Z 282.592,A -85,B 0,C 180,E1 -3744.532,E2 -3744.532} C_VEL
LIN {X 0,Y 545.077,Z 282.586,A -85,B 0,C 180,E1 -3747.212,E2 -3747.212} C_VEL
LIN {X 0,Y 545.061,Z 282.583,A -85,B 0,C 180,E1 -3749.81,E2 -3749.81} C_VEL
LIN {X 0,Y 545.084,Z 282.582,A -85,B 0,C 180,E1 -3752.344,E2 -3752.344} C_VEL
LIN {X 0,Y 545.112,Z 282.584,A -85,B 0,C 180,E1 -3754.82,E2 -3754.82} C_VEL
LIN {X 0,Y 545.039,Z 282.594,A -85,B 0,C 180,E1 -3757.242,E2 -3757.242} C_VEL
LIN {X 0,Y 545.115,Z 282.577,A -85,B 0,C 180,E1 -3760.415,E2 -3760.415} C_VEL
LIN {X 0,Y 545.067,Z 282.589,A -85,B 0,C 180,E1 -3763.521,E2 -3763.521} C_VEL
LIN {X 0,Y 545.089,Z 282.583,A -85,B 0,C 180,E1 -3765.82,E2 -3765.82} C_VEL
LIN {X 0,Y 545.112,Z 282.579,A -85,B 0,C 180,E1 -3768.849,E2 -3768.849} C_VEL
LIN {X 0,Y 545.125,Z 282.58,A -85,B 0,C 180,E1 -3771.847,E2 -3771.847} C_VEL
LIN {X 0,Y 545.2,Z 282.567,A -85,B 0,C 180,E1 -3774.823,E2 -3774.823} C_VEL
LIN {X 0,Y 545.186,Z 282.576,A -85,B 0,C 180,E1 -3777.784,E2 -3777.784} C_VEL
LIN {X 0,Y 545.204,Z 282.566,A -85,B 0,C 180,E1 -3780.739,E2 -3780.739} C_VEL
LIN {X 0,Y 545.165,Z 282.571,A -85,B 0,C 180,E1 -3782.956,E2 -3782.956} C_VEL
LIN {X 0,Y 545.16,Z 282.581,A -85,B 0,C 180,E1 -3785.92,E2 -3785.92} C_VEL
LIN {X 0,Y 545.111,Z 282.577,A -85,B 0,C 180,E1 -3788.9,E2 -3788.9} C_VEL
LIN {X 0,Y 545.129,Z 282.583,A -85,B 0,C 180,E1 -3791.905,E2 -3791.905} C_VEL
LIN {X 0,Y 545.076,Z 282.582,A -85,B 0,C 180,E1 -3794.944,E2 -3794.944} C_VEL
LIN {X 0,Y 545.065,Z 282.59,A -85,B 0,C 180,E1 -3798.027,E2 -3798.027} C_VEL
LIN {X 0,Y 545.087,Z 282.589,A -85,B 0,C 180,E1 -3800.373,E2 -3800.373} C_VEL
LIN {X 0,Y 545.074,Z 282.582,A -85,B 0,C 180,E1 -3803.56,E2 -3803.56} C_VEL
LIN {X 0,Y 545.071,Z 282.586,A -85,B 0,C 180,E1 -3806.001,E2 -3806.001} C_VEL
LIN {X 0,Y 545.064,Z 282.589,A -85,B 0,C 180,E1 -3808.745,E2 -3808.745} C_VEL
LIN {X 0,Y 545.054,Z 282.584,A -85,B 0,C 180,E1 -3811.679,E2 -3811.679} C_VEL
LIN {X 0,Y 545.058,Z 282.593,A -85,B 0,C 180,E1 -3814.565,E2 -3814.565} C_VEL
LIN {X 0,Y 545.059,Z 282.59,A -85,B 0,C 180,E1 -3816.989,E2 -3816.989} C_VEL
LIN {X 0,Y 544.35,Z 282.675,A -85,B 0,C 180,E1 -3817.605,E2 -3817.605} C_VEL
LIN {X 0,Y 541.482,Z 283.037,A -85,B 0,C 180,E1 -3818.606,E2 -3818.606} C_VEL
LIN {X 0,Y 539.089,Z 283.33,A -85,B 0,C 180,E1 -3819.412,E2 -3819.412} C_VEL
LIN {X 0,Y 538.073,Z 283.455,A -85,B 0,C 180,E1 -3820.034,E2 -3820.034} C_VEL
LIN {X 0,Y 537.995,Z 283.466,A -85,B 0,C 180,E1 -3820.244,E2 -3820.244} C_VEL
LIN {X 0,Y 537.978,Z 283.475,A -85,B 0,C 180,E1 -3822.983,E2 -3822.983} C_VEL
LIN {X 0,Y 538.016,Z 283.461,A -85,B 0,C 180,E1 -3825.928,E2 -3825.928} C_VEL
LIN {X 0,Y 538.001,Z 283.471,A -85,B 0,C 180,E1 -3829.221,E2 -3829.221} C_VEL
LIN {X 0,Y 537.986,Z 283.465,A -85,B 0,C 180,E1 -3832.123,E2 -3832.123} C_VEL
LIN {X 0,Y 537.993,Z 283.469,A -85,B 0,C 180,E1 -3834.916,E2 -3834.916} C_VEL
LIN {X 0,Y 538.012,Z 283.466,A -85,B 0,C 180,E1 -3837.618,E2 -3837.618} C_VEL
LIN {X 0,Y 537.998,Z 283.463,A -85,B 0,C 180,E1 -3840.238,E2 -3840.238} C_VEL
LIN {X 0,Y 538.002,Z 283.464,A -85,B 0,C 180,E1 -3842.793,E2 -3842.793} C_VEL
LIN {X 0,Y 537.98,Z 283.472,A -85,B 0,C 180,E1 -3845.29,E2 -3845.29} C_VEL
LIN {X 0,Y 538.018,Z 283.464,A -85,B 0,C 180,E1 -3848.043,E2 -3848.043} C_VEL
LIN {X 0,Y 538.044,Z 283.46,A -85,B 0,C 180,E1 -3850.147,E2 -3850.147} C_VEL
LIN {X 0,Y 537.989,Z 283.468,A -85,B 0,C 180,E1 -3853.298,E2 -3853.298} C_VEL
LIN {X 0,Y 538.063,Z 283.463,A -85,B 0,C 180,E1 -3855.631,E2 -3855.631} C_VEL
LIN {X 0,Y 538.027,Z 283.46,A -85,B 0,C 180,E1 -3858.701,E2 -3858.701} C_VEL
LIN {X 0,Y 538.037,Z 283.465,A -85,B 0,C 180,E1 -3861.739,E2 -3861.739} C_VEL
LIN {X 0,Y 538.122,Z 283.449,A -85,B 0,C 180,E1 -3864.755,E2 -3864.755} C_VEL
LIN {X 0,Y 538.163,Z 283.447,A -85,B 0,C 180,E1 -3867.755,E2 -3867.755} C_VEL
LIN {X 0,Y 538.162,Z 283.45,A -85,B 0,C 180,E1 -3870,E2 -3870} C_VEL
LIN {X 0,Y 538.083,Z 283.453,A -85,B 0,C 180,E1 -3872.995,E2 -3872.995} C_VEL
LIN {X 0,Y 538.082,Z 283.458,A -85,B 0,C 180,E1 -3875.998,E2 -3875.998} C_VEL
LIN {X 0,Y 538.024,Z 283.462,A -85,B 0,C 180,E1 -3879.019,E2 -3879.019} C_VEL
LIN {X 0,Y 538.008,Z 283.465,A -85,B 0,C 180,E1 -3882.065,E2 -3882.065} C_VEL
LIN {X 0,Y 537.989,Z 283.466,A -85,B 0,C 180,E1 -3885.146,E2 -3885.146} C_VEL
LIN {X 0,Y 538,Z 283.467,A -85,B 0,C 180,E1 -3888.272,E2 -3888.272} C_VEL
LIN {X 0,Y 537.992,Z 283.473,A -85,B 0,C 180,E1 -3890.654,E2 -3890.654} C_VEL
LIN {X 0,Y 537.99,Z 283.472,A -85,B 0,C 180,E1 -3893.073,E2 -3893.073} C_VEL
LIN {X 0,Y 537.967,Z 283.471,A -85,B 0,C 180,E1 -3895.654,E2 -3895.654} C_VEL
LIN {X 0,Y 538.038,Z 283.566,A -85,B 0,C 180,E1 -3897.486,E2 -3897.486} C_VEL
LIN {X 0,Y 538.463,Z 288.519,A -85,B 0,C 180,E1 -3898.451,E2 -3898.451} C_VEL
LIN {X 0,Y 538.268,Z 303.366,A -85,B 0,C 180,E1 -3901.266,E2 -3901.266} C_VEL
LIN {X 0,Y 538.199,Z 308.872,A -85,B 0,C 180,E1 -3902.305,E2 -3902.305} C_VEL
LIN {X 0,Y 539.641,Z 317.288,A -85,B 0,C 180,E1 -3902.467,E2 -3902.467} C_VEL
LIN {X 0,Y 539.314,Z 415.636,A -85,B 0,C 180,E1 -3903.805,E2 -3903.805} C_VEL
LIN {X 0,Y 539.115,Z 429.173,A -85,B 0,C 180,E1 -3904.148,E2 -3904.148} C_VEL
LIN {X 0,Y 538.998,Z 439.51,A -85,B 0,C 180,E1 -3904.529,E2 -3904.529} C_VEL
LIN {X 0,Y 538.746,Z 450.943,A -85,B 0,C 180,E1 -3905.086,E2 -3905.086} C_VEL
LIN {X 0,Y 538.56,Z 459.691,A -85,B 0,C 180,E1 -3905.615,E2 -3905.615} C_VEL
LIN {X 0,Y 538.372,Z 469.253,A -85,B 0,C 180,E1 -3906.323,E2 -3906.323} C_VEL
LIN {X 0,Y 538.188,Z 477.483,A -85,B 0,C 180,E1 -3907.052,E2 -3907.052} C_VEL
LIN {X 0,Y 538.025,Z 485.275,A -85,B 0,C 180,E1 -3907.875,E2 -3907.875} C_VEL
LIN {X 0,Y 537.923,Z 491.008,A -85,B 0,C 180,E1 -3908.576,E2 -3908.576} C_VEL
LIN {X 0,Y 537.78,Z 497.712,A -85,B 0,C 180,E1 -3909.552,E2 -3909.552} C_VEL
LIN {X 0,Y 537.661,Z 504.097,A -85,B 0,C 180,E1 -3910.699,E2 -3910.699} C_VEL
LIN {X 0,Y 537.602,Z 509.109,A -85,B 0,C 180,E1 -3911.827,E2 -3911.827} C_VEL
LIN {X 0,Y 537.567,Z 512.938,A -85,B 0,C 180,E1 -3912.934,E2 -3912.934} C_VEL
LIN {X 0,Y 537.516,Z 515.734,A -85,B 0,C 180,E1 -3914.017,E2 -3914.017} C_VEL
LIN {X 0,Y 537.495,Z 517.627,A -85,B 0,C 180,E1 -3915.083,E2 -3915.083} C_VEL
LIN {X 0,Y 537.47,Z 518.705,A -85,B 0,C 180,E1 -3916.129,E2 -3916.129} C_VEL
LIN {X 0,Y 537.471,Z 519.03,A -85,B 0,C 180,E1 -3917.159,E2 -3917.159} C_VEL
LIN {X 0,Y 537.466,Z 518.592,A -85,B 0,C 180,E1 -3918.189,E2 -3918.189} C_VEL
LIN {X 0,Y 537.467,Z 517.224,A -85,B 0,C 180,E1 -3919.325,E2 -3919.325} C_VEL
LIN {X 0,Y 537.498,Z 514.866,A -85,B 0,C 180,E1 -3920.484,E2 -3920.484} C_VEL
LIN {X 0,Y 537.558,Z 511.384,A -85,B 0,C 180,E1 -3921.669,E2 -3921.669} C_VEL
LIN {X 0,Y 537.622,Z 506.544,A -85,B 0,C 180,E1 -3922.884,E2 -3922.884} C_VEL
LIN {X 0,Y 537.727,Z 501.033,A -85,B 0,C 180,E1 -3923.974,E2 -3923.974} C_VEL
LIN {X 0,Y 537.812,Z 495.361,A -85,B 0,C 180,E1 -3924.901,E2 -3924.901} C_VEL
LIN {X 0,Y 537.954,Z 488.607,A -85,B 0,C 180,E1 -3925.822,E2 -3925.822} C_VEL
LIN {X 0,Y 538.114,Z 480.564,A -85,B 0,C 180,E1 -3926.733,E2 -3926.733} C_VEL
LIN {X 0,Y 538.303,Z 472.179,A -85,B 0,C 180,E1 -3927.525,E2 -3927.525} C_VEL
LIN {X 0,Y 538.478,Z 462.565,A -85,B 0,C 180,E1 -3928.277,E2 -3928.277} C_VEL
LIN {X 0,Y 538.718,Z 452.711,A -85,B 0,C 180,E1 -3928.905,E2 -3928.905} C_VEL
LIN {X 0,Y 538.898,Z 443.136,A -85,B 0,C 180,E1 -3929.399,E2 -3929.399} C_VEL
LIN {X 0,Y 539.056,Z 432.838,A -85,B 0,C 180,E1 -3929.817,E2 -3929.817} C_VEL
LIN {X 0,Y 539.172,Z 422.293,A -85,B 0,C 180,E1 -3930.134,E2 -3930.134} C_VEL
LIN {X 0,Y 539.278,Z 410.273,A -85,B 0,C 180,E1 -3930.375,E2 -3930.375} C_VEL
LIN {X 0,Y 539.514,Z 316.431,A -85,B 0,C 180,E1 -3931.636,E2 -3931.636} C_VEL
LIN {X 0,Y 538.181,Z 308.617,A -85,B 0,C 180,E1 -3931.799,E2 -3931.799} C_VEL
LIN {X 0,Y 538.228,Z 293.977,A -85,B 0,C 180,E1 -3934.287,E2 -3934.287} C_VEL
LIN {X 0,Y 538.144,Z 283.452,A -85,B 0,C 180,E1 -3936.026,E2 -3936.026} C_VEL
LIN {X 0,Y 538.04,Z 283.468,A -85,B 0,C 180,E1 -3939.348,E2 -3939.348} C_VEL
LIN {X 0,Y 538.038,Z 283.461,A -85,B 0,C 180,E1 -3942.467,E2 -3942.467} C_VEL
LIN {X 0,Y 538.066,Z 283.465,A -85,B 0,C 180,E1 -3945.63,E2 -3945.63} C_VEL
LIN {X 0,Y 538.079,Z 283.454,A -85,B 0,C 180,E1 -3948.701,E2 -3948.701} C_VEL
LIN {X 0,Y 538.08,Z 283.463,A -85,B 0,C 180,E1 -3951.739,E2 -3951.739} C_VEL
LIN {X 0,Y 538.119,Z 283.455,A -85,B 0,C 180,E1 -3954.002,E2 -3954.002} C_VEL
LIN {X 0,Y 538.138,Z 283.447,A -85,B 0,C 180,E1 -3957.005,E2 -3957.005} C_VEL
LIN {X 0,Y 538.174,Z 283.45,A -85,B 0,C 180,E1 -3960,E2 -3960} C_VEL
LIN {X 0,Y 538.138,Z 283.446,A -85,B 0,C 180,E1 -3962.994,E2 -3962.994} C_VEL
LIN {X 0,Y 538.113,Z 283.458,A -85,B 0,C 180,E1 -3965.997,E2 -3965.997} C_VEL
LIN {X 0,Y 538.062,Z 283.456,A -85,B 0,C 180,E1 -3969.018,E2 -3969.018} C_VEL
LIN {X 0,Y 538.084,Z 283.459,A -85,B 0,C 180,E1 -3972.062,E2 -3972.062} C_VEL
LIN {X 0,Y 538.047,Z 283.459,A -85,B 0,C 180,E1 -3975.144,E2 -3975.144} C_VEL
LIN {X 0,Y 538.027,Z 283.465,A -85,B 0,C 180,E1 -3978.27,E2 -3978.27} C_VEL
LIN {X 0,Y 538.039,Z 283.466,A -85,B 0,C 180,E1 -3980.651,E2 -3980.651} C_VEL
LIN {X 0,Y 538.004,Z 283.463,A -85,B 0,C 180,E1 -3983.888,E2 -3983.888} C_VEL
LIN {X 0,Y 538.043,Z 283.461,A -85,B 0,C 180,E1 -3986.367,E2 -3986.367} C_VEL
LIN {X 0,Y 538.032,Z 283.469,A -85,B 0,C 180,E1 -3988.933,E2 -3988.933} C_VEL
LIN {X 0,Y 538.011,Z 283.461,A -85,B 0,C 180,E1 -3991.887,E2 -3991.887} C_VEL
LIN {X 0,Y 538.01,Z 283.465,A -85,B 0,C 180,E1 -3994.617,E2 -3994.617} C_VEL
LIN {X 0,Y 538.006,Z 283.471,A -85,B 0,C 180,E1 -3997.17,E2 -3997.17} C_VEL
LIN {X 0,Y 538.024,Z 283.462,A -85,B 0,C 180,E1 -3999.797,E2 -3999.797} C_VEL
LIN {X 0,Y 538.02,Z 283.464,A -85,B 0,C 180,E1 -4002.786,E2 -4002.786} C_VEL
LIN {X 0,Y 538.02,Z 283.464,A -85,B 0,C 180,E1 -4005.927,E2 -4005.927} C_VEL
LIN {X 0,Y 538.032,Z 283.46,A -85,B 0,C 180,E1 -4008.227,E2 -4008.227} C_VEL
LIN {X 0,Y 538.014,Z 283.466,A -85,B 0,C 180,E1 -4011.169,E2 -4011.169} C_VEL
LIN {X 0,Y 537.996,Z 283.47,A -85,B 0,C 180,E1 -4014.089,E2 -4014.089} C_VEL
LIN {X 0,Y 538.033,Z 283.462,A -85,B 0,C 180,E1 -4016.727,E2 -4016.727} C_VEL
LIN {X 0,Y 538.029,Z 283.467,A -85,B 0,C 180,E1 -4019.556,E2 -4019.556} C_VEL
LIN {X 0,Y 538.04,Z 283.469,A -85,B 0,C 180,E1 -4021.95,E2 -4021.95} C_VEL
LIN {X 0,Y 538.066,Z 283.463,A -85,B 0,C 180,E1 -4024.467,E2 -4024.467} C_VEL
LIN {X 0,Y 538.071,Z 283.619,A -85,B 0,C 180,E1 -4025.953,E2 -4025.953} C_VEL
LIN {X 0,Y 539.164,Z 290.197,A -85,B 0,C 180,E1 -4026.98,E2 -4026.98} C_VEL
LIN {X 0,Y 538.875,Z 309.681,A -85,B 0,C 180,E1 -4029.888,E2 -4029.888} C_VEL
LIN {X 0,Y 538.532,Z 330.19,A -85,B 0,C 180,E1 -4032.924,E2 -4032.924} C_VEL
LIN {X 0,Y 538.323,Z 346.009,A -85,B 0,C 180,E1 -4035.237,E2 -4035.237} C_VEL
LIN {X 0,Y 539.636,Z 355.888,A -85,B 0,C 180,E1 -4035.419,E2 -4035.419} C_VEL
LIN {X 0,Y 539.25,Z 455.257,A -85,B 0,C 180,E1 -4036.768,E2 -4036.768} C_VEL
LIN {X 0,Y 539.125,Z 468.322,A -85,B 0,C 180,E1 -4037.1,E2 -4037.1} C_VEL
LIN {X 0,Y 538.9,Z 480.953,A -85,B 0,C 180,E1 -4037.573,E2 -4037.573} C_VEL
LIN {X 0,Y 538.724,Z 492.878,A -85,B 0,C 180,E1 -4038.184,E2 -4038.184} C_VEL
LIN {X 0,Y 538.504,Z 503.847,A -85,B 0,C 180,E1 -4038.901,E2 -4038.901} C_VEL
LIN {X 0,Y 538.254,Z 514.337,A -85,B 0,C 180,E1 -4039.752,E2 -4039.752} C_VEL
LIN {X 0,Y 538.067,Z 522.914,A -85,B 0,C 180,E1 -4040.603,E2 -4040.603} C_VEL
LIN {X 0,Y 537.913,Z 530.825,A -85,B 0,C 180,E1 -4041.547,E2 -4041.547} C_VEL
LIN {X 0,Y 537.755,Z 538.548,A -85,B 0,C 180,E1 -4042.679,E2 -4042.679} C_VEL
LIN {X 0,Y 537.696,Z 545.665,A -85,B 0,C 180,E1 -4043.998,E2 -4043.998} C_VEL
LIN {X 0,Y 537.54,Z 550.371,A -85,B 0,C 180,E1 -4045.125,E2 -4045.125} C_VEL
LIN {X 0,Y 537.591,Z 553.956,A -85,B 0,C 180,E1 -4046.252,E2 -4046.252} C_VEL
LIN {X 0,Y 537.551,Z 555.805,A -85,B 0,C 180,E1 -4047.002,E2 -4047.002} C_VEL
LIN {X 0,Y 537.451,Z 558.181,A -85,B 0,C 180,E1 -4048.501,E2 -4048.501} C_VEL
LIN {X 0,Y 537.442,Z 559,A -85,B 0,C 180,E1 -4050,E2 -4050} C_VEL
LIN {X 0,Y 537.451,Z 558.183,A -85,B 0,C 180,E1 -4051.498,E2 -4051.498} C_VEL
LIN {X 0,Y 537.551,Z 555.811,A -85,B 0,C 180,E1 -4052.997,E2 -4052.997} C_VEL
LIN {X 0,Y 537.603,Z 552.896,A -85,B 0,C 180,E1 -4054.123,E2 -4054.123} C_VEL
LIN {X 0,Y 537.587,Z 548.949,A -85,B 0,C 180,E1 -4055.25,E2 -4055.25} C_VEL
LIN {X 0,Y 537.642,Z 544.101,A -85,B 0,C 180,E1 -4056.326,E2 -4056.326} C_VEL
LIN {X 0,Y 537.771,Z 537.392,A -85,B 0,C 180,E1 -4057.509,E2 -4057.509} C_VEL
LIN {X 0,Y 537.941,Z 529.347,A -85,B 0,C 180,E1 -4058.641,E2 -4058.641} C_VEL
LIN {X 0,Y 538.114,Z 521.146,A -85,B 0,C 180,E1 -4059.585,E2 -4059.585} C_VEL
LIN {X 0,Y 538.345,Z 511.145,A -85,B 0,C 180,E1 -4060.53,E2 -4060.53} C_VEL
LIN {X 0,Y 538.597,Z 501.275,A -85,B 0,C 180,E1 -4061.287,E2 -4061.287} C_VEL
LIN {X 0,Y 538.736,Z 490.045,A -85,B 0,C 180,E1 -4061.978,E2 -4061.978} C_VEL
LIN {X 0,Y 538.933,Z 477.624,A -85,B 0,C 180,E1 -4062.568,E2 -4062.568} C_VEL
LIN {X 0,Y 539.146,Z 464.476,A -85,B 0,C 180,E1 -4063.018,E2 -4063.018} C_VEL
LIN {X 0,Y 539.334,Z 451.305,A -85,B 0,C 180,E1 -4063.301,E2 -4063.301} C_VEL
LIN {X 0,Y 539.566,Z 354.632,A -85,B 0,C 180,E1 -4064.6,E2 -4064.6} C_VEL
LIN {X 0,Y 538.336,Z 346.239,A -85,B 0,C 180,E1 -4064.761,E2 -4064.761} C_VEL
LIN {X 0,Y 538.718,Z 323.865,A -85,B 0,C 180,E1 -4068.085,E2 -4068.085} C_VEL
LIN {X 0,Y 539.036,Z 305.746,A -85,B 0,C 180,E1 -4070.81,E2 -4070.81} C_VEL
LIN {X 0,Y 539.373,Z 291.362,A -85,B 0,C 180,E1 -4073.01,E2 -4073.01} C_VEL
LIN {X 0,Y 538.033,Z 283.468,A -85,B 0,C 180,E1 -4074.322,E2 -4074.322} C_VEL
LIN {X 0,Y 538.063,Z 283.458,A -85,B 0,C 180,E1 -4077.203,E2 -4077.203} C_VEL
LIN {X 0,Y 538.016,Z 283.467,A -85,B 0,C 180,E1 -4079.76,E2 -4079.76} C_VEL
LIN {X 0,Y 538.017,Z 283.468,A -85,B 0,C 180,E1 -4082.382,E2 -4082.382} C_VEL
LIN {X 0,Y 537.997,Z 283.464,A -85,B 0,C 180,E1 -4085.084,E2 -4085.084} C_VEL
LIN {X 0,Y 537.99,Z 283.468,A -85,B 0,C 180,E1 -4087.877,E2 -4087.877} C_VEL
LIN {X 0,Y 538.046,Z 283.461,A -85,B 0,C 180,E1 -4090.775,E2 -4090.775} C_VEL
LIN {X 0,Y 538.027,Z 283.464,A -85,B 0,C 180,E1 -4094.074,E2 -4094.074} C_VEL
LIN {X 0,Y 538.019,Z 283.462,A -85,B 0,C 180,E1 -4097.214,E2 -4097.214} C_VEL
LIN {X 0,Y 538.025,Z 283.463,A -85,B 0,C 180,E1 -4100.203,E2 -4100.203} C_VEL
LIN {X 0,Y 538.024,Z 283.465,A -85,B 0,C 180,E1 -4103.067,E2 -4103.067} C_VEL
LIN {X 0,Y 538.02,Z 283.461,A -85,B 0,C 180,E1 -4105.827,E2 -4105.827} C_VEL
LIN {X 0,Y 538.019,Z 283.465,A -85,B 0,C 180,E1 -4108.499,E2 -4108.499} C_VEL
LIN {X 0,Y 538.055,Z 283.464,A -85,B 0,C 180,E1 -4111.1,E2 -4111.1} C_VEL
LIN {X 0,Y 538.037,Z 283.46,A -85,B 0,C 180,E1 -4113.633,E2 -4113.633} C_VEL
LIN {X 0,Y 538.017,Z 283.461,A -85,B 0,C 180,E1 -4116.118,E2 -4116.118} C_VEL
LIN {X 0,Y 538.034,Z 283.466,A -85,B 0,C 180,E1 -4119.348,E2 -4119.348} C_VEL
LIN {X 0,Y 538.048,Z 283.458,A -85,B 0,C 180,E1 -4122.517,E2 -4122.517} C_VEL
LIN {X 0,Y 538.058,Z 283.461,A -85,B 0,C 180,E1 -4125.631,E2 -4125.631} C_VEL
LIN {X 0,Y 538.071,Z 283.455,A -85,B 0,C 180,E1 -4128.702,E2 -4128.702} C_VEL
LIN {X 0,Y 538.082,Z 283.459,A -85,B 0,C 180,E1 -4131.74,E2 -4131.74} C_VEL
LIN {X 0,Y 538.157,Z 283.444,A -85,B 0,C 180,E1 -4134.755,E2 -4134.755} C_VEL
LIN {X 0,Y 538.158,Z 283.452,A -85,B 0,C 180,E1 -4137.755,E2 -4137.755} C_VEL
LIN {X 0,Y 538.175,Z 283.441,A -85,B 0,C 180,E1 -4140.748,E2 -4140.748} C_VEL
LIN {X 0,Y 538.132,Z 283.447,A -85,B 0,C 180,E1 -4142.995,E2 -4142.995} C_VEL
LIN {X 0,Y 538.111,Z 283.458,A -85,B 0,C 180,E1 -4145.998,E2 -4145.998} C_VEL
LIN {X 0,Y 538.062,Z 283.455,A -85,B 0,C 180,E1 -4149.018,E2 -4149.018} C_VEL
LIN {X 0,Y 538.077,Z 283.464,A -85,B 0,C 180,E1 -4152.063,E2 -4152.063} C_VEL
LIN {X 0,Y 538.037,Z 283.458,A -85,B 0,C 180,E1 -4155.144,E2 -4155.144} C_VEL
LIN {X 0,Y 538.019,Z 283.47,A -85,B 0,C 180,E1 -4158.271,E2 -4158.271} C_VEL
LIN {X 0,Y 538.032,Z 283.463,A -85,B 0,C 180,E1 -4160.652,E2 -4160.652} C_VEL
LIN {X 0,Y 537.997,Z 283.466,A -85,B 0,C 180,E1 -4163.889,E2 -4163.889} C_VEL
LIN {X 0,Y 538.031,Z 283.468,A -85,B 0,C 180,E1 -4166.368,E2 -4166.368} C_VEL
LIN {X 0,Y 538.025,Z 283.463,A -85,B 0,C 180,E1 -4168.934,E2 -4168.934} C_VEL
LIN {X 0,Y 538.006,Z 283.463,A -85,B 0,C 180,E1 -4171.888,E2 -4171.888} C_VEL
LIN {X 0,Y 538.008,Z 283.472,A -85,B 0,C 180,E1 -4174.618,E2 -4174.618} C_VEL
LIN {X 0,Y 538,Z 283.466,A -85,B 0,C 180,E1 -4177.171,E2 -4177.171} C_VEL
LIN {X 0,Y 538.007,Z 283.462,A -85,B 0,C 180,E1 -4179.799,E2 -4179.799} C_VEL
LIN {X 0,Y 537.995,Z 283.466,A -85,B 0,C 180,E1 -4180.244,E2 -4180.244} C_VEL
LIN {X 0,Y 537.338,Z 283.556,A -85,B 0,C 180,E1 -4180.869,E2 -4180.869} C_VEL
LIN {X 0,Y 534.484,Z 283.91,A -85,B 0,C 180,E1 -4181.884,E2 -4181.884} C_VEL
LIN {X 0,Y 532.063,Z 284.21,A -85,B 0,C 180,E1 -4182.702,E2 -4182.702} C_VEL
LIN {X 0,Y 531.02,Z 284.337,A -85,B 0,C 180,E1 -4183.333,E2 -4183.333} C_VEL
LIN {X 0,Y 530.934,Z 284.345,A -85,B 0,C 180,E1 -4183.546,E2 -4183.546} C_VEL
LIN {X 0,Y 530.943,Z 284.345,A -85,B 0,C 180,E1 -4186.504,E2 -4186.504} C_VEL
LIN {X 0,Y 530.949,Z 284.344,A -85,B 0,C 180,E1 -4189.565,E2 -4189.565} C_VEL
LIN {X 0,Y 530.964,Z 284.341,A -85,B 0,C 180,E1 -4192.578,E2 -4192.578} C_VEL
LIN {X 0,Y 530.978,Z 284.347,A -85,B 0,C 180,E1 -4195.31,E2 -4195.31} C_VEL
LIN {X 0,Y 530.958,Z 284.341,A -85,B 0,C 180,E1 -4198.032,E2 -4198.032} C_VEL
LIN {X 0,Y 530.964,Z 284.342,A -85,B 0,C 180,E1 -4200.88,E2 -4200.88} C_VEL
LIN {X 0,Y 530.949,Z 284.348,A -85,B 0,C 180,E1 -4203.254,E2 -4203.254} C_VEL
LIN {X 0,Y 530.955,Z 284.344,A -85,B 0,C 180,E1 -4205.97,E2 -4205.97} C_VEL
LIN {X 0,Y 531,Z 284.337,A -85,B 0,C 180,E1 -4209.063,E2 -4209.063} C_VEL
LIN {X 0,Y 530.961,Z 284.347,A -85,B 0,C 180,E1 -4211.478,E2 -4211.478} C_VEL
LIN {X 0,Y 530.989,Z 284.337,A -85,B 0,C 180,E1 -4214.651,E2 -4214.651} C_VEL
LIN {X 0,Y 531.012,Z 284.343,A -85,B 0,C 180,E1 -4217.775,E2 -4217.775} C_VEL
LIN {X 0,Y 530.995,Z 284.336,A -85,B 0,C 180,E1 -4220.862,E2 -4220.862} C_VEL
LIN {X 0,Y 531.046,Z 284.338,A -85,B 0,C 180,E1 -4223.923,E2 -4223.923} C_VEL
LIN {X 0,Y 531.029,Z 284.332,A -85,B 0,C 180,E1 -4226.966,E2 -4226.966} C_VEL
LIN {X 0,Y 531.018,Z 284.337,A -85,B 0,C 180,E1 -4228.484,E2 -4228.484} C_VEL
LIN {X 0,Y 531.131,Z 284.326,A -85,B 0,C 180,E1 -4230,E2 -4230} C_VEL
LIN {X 0,Y 531.131,Z 284.329,A -85,B 0,C 180,E1 -4232.275,E2 -4232.275} C_VEL
LIN {X 0,Y 531.082,Z 284.325,A -85,B 0,C 180,E1 -4235.316,E2 -4235.316} C_VEL
LIN {X 0,Y 530.983,Z 284.347,A -85,B 0,C 180,E1 -4238.372,E2 -4238.372} C_VEL
LIN {X 0,Y 531.009,Z 284.334,A -85,B 0,C 180,E1 -4241.646,E2 -4241.646} C_VEL
LIN {X 0,Y 530.967,Z 284.344,A -85,B 0,C 180,E1 -4244.927,E2 -4244.927} C_VEL
LIN {X 0,Y 530.976,Z 284.338,A -85,B 0,C 180,E1 -4247.724,E2 -4247.724} C_VEL
LIN {X 0,Y 530.964,Z 284.348,A -85,B 0,C 180,E1 -4250.94,E2 -4250.94} C_VEL
LIN {X 0,Y 530.955,Z 284.343,A -85,B 0,C 180,E1 -4254.031,E2 -4254.031} C_VEL
LIN {X 0,Y 531.011,Z 284.475,A -85,B 0,C 180,E1 -4257.377,E2 -4257.377} C_VEL
LIN {X 0,Y 531.507,Z 288.68,A -85,B 0,C 180,E1 -4258.211,E2 -4258.211} C_VEL
LIN {X 0,Y 531.288,Z 303.527,A -85,B 0,C 180,E1 -4261.058,E2 -4261.058} C_VEL
LIN {X 0,Y 531.228,Z 309.238,A -85,B 0,C 180,E1 -4262.117,E2 -4262.117} C_VEL
LIN {X 0,Y 532.759,Z 317.931,A -85,B 0,C 180,E1 -4262.282,E2 -4262.282} C_VEL
LIN {X 0,Y 532.42,Z 415.875,A -85,B 0,C 180,E1 -4263.635,E2 -4263.635} C_VEL
LIN {X 0,Y 532.21,Z 429.439,A -85,B 0,C 180,E1 -4263.982,E2 -4263.982} C_VEL
LIN {X 0,Y 532.032,Z 440.981,A -85,B 0,C 180,E1 -4264.423,E2 -4264.423} C_VEL
LIN {X 0,Y 531.776,Z 451.948,A -85,B 0,C 180,E1 -4264.975,E2 -4264.975} C_VEL
LIN {X 0,Y 531.581,Z 461.416,A -85,B 0,C 180,E1 -4265.572,E2 -4265.572} C_VEL
LIN {X 0,Y 531.376,Z 469.888,A -85,B 0,C 180,E1 -4266.216,E2 -4266.216} C_VEL
LIN {X 0,Y 531.165,Z 478.651,A -85,B 0,C 180,E1 -4267.015,E2 -4267.015} C_VEL
LIN {X 0,Y 531.014,Z 486.415,A -85,B 0,C 180,E1 -4267.863,E2 -4267.863} C_VEL
LIN {X 0,Y 530.824,Z 493.596,A -85,B 0,C 180,E1 -4268.799,E2 -4268.799} C_VEL
LIN {X 0,Y 530.67,Z 500.05,A -85,B 0,C 180,E1 -4269.813,E2 -4269.813} C_VEL
LIN {X 0,Y 530.559,Z 506.036,A -85,B 0,C 180,E1 -4270.97,E2 -4270.97} C_VEL
LIN {X 0,Y 530.498,Z 510.689,A -85,B 0,C 180,E1 -4272.107,E2 -4272.107} C_VEL
LIN {X 0,Y 530.433,Z 515.093,A -85,B 0,C 180,E1 -4273.549,E2 -4273.549} C_VEL
LIN {X 0,Y 530.423,Z 517.266,A -85,B 0,C 180,E1 -4274.607,E2 -4274.607} C_VEL
LIN {X 0,Y 530.393,Z 518.658,A -85,B 0,C 180,E1 -4275.687,E2 -4275.687} C_VEL
LIN {X 0,Y 530.35,Z 519.252,A -85,B 0,C 180,E1 -4276.789,E2 -4276.789} C_VEL
LIN {X 0,Y 530.373,Z 519.009,A -85,B 0,C 180,E1 -4277.907,E2 -4277.907} C_VEL
LIN {X 0,Y 530.382,Z 517.884,A -85,B 0,C 180,E1 -4279.052,E2 -4279.052} C_VEL
LIN {X 0,Y 530.418,Z 515.184,A -85,B 0,C 180,E1 -4280.506,E2 -4280.506} C_VEL
LIN {X 0,Y 530.488,Z 512.42,A -85,B 0,C 180,E1 -4281.489,E2 -4281.489} C_VEL
LIN {X 0,Y 530.551,Z 508.237,A -85,B 0,C 180,E1 -4282.636,E2 -4282.636} C_VEL
LIN {X 0,Y 530.655,Z 502.307,A -85,B 0,C 180,E1 -4283.89,E2 -4283.89} C_VEL
LIN {X 0,Y 530.767,Z 495.525,A -85,B 0,C 180,E1 -4285.019,E2 -4285.019} C_VEL
LIN {X 0,Y 530.95,Z 488.379,A -85,B 0,C 180,E1 -4285.996,E2 -4285.996} C_VEL
LIN {X 0,Y 531.154,Z 480.131,A -85,B 0,C 180,E1 -4286.929,E2 -4286.929} C_VEL
LIN {X 0,Y 531.307,Z 471.622,A -85,B 0,C 180,E1 -4287.732,E2 -4287.732} C_VEL
LIN {X 0,Y 531.5,Z 463.139,A -85,B 0,C 180,E1 -4288.401,E2 -4288.401} C_VEL
LIN {X 0,Y 531.771,Z 453.149,A -85,B 0,C 180,E1 -4289.049,E2 -4289.049} C_VEL
LIN {X 0,Y 531.991,Z 442.357,A -85,B 0,C 180,E1 -4289.607,E2 -4289.607} C_VEL
LIN {X 0,Y 532.151,Z 431.349,A -85,B 0,C 180,E1 -4290.044,E2 -4290.044} C_VEL
LIN {X 0,Y 532.303,Z 419.433,A -85,B 0,C 180,E1 -4290.381,E2 -4290.381} C_VEL
LIN {X 0,Y 532.391,Z 402.652,A -85,B 0,C 180,E1 -4290.654,E2 -4290.654} C_VEL
LIN {X 0,Y 532.775,Z 317.873,A -85,B 0,C 180,E1 -4291.809,E2 -4291.809} C_VEL
LIN {X 0,Y 531.167,Z 308.684,A -85,B 0,C 180,E1 -4291.998,E2 -4291.998} C_VEL
LIN {X 0,Y 531.189,Z 291.118,A -85,B 0,C 180,E1 -4294.951,E2 -4294.951} C_VEL
LIN {X 0,Y 531.119,Z 284.328,A -85,B 0,C 180,E1 -4296.077,E2 -4296.077} C_VEL
LIN {X 0,Y 531.027,Z 284.336,A -85,B 0,C 180,E1 -4299.873,E2 -4299.873} C_VEL
LIN {X 0,Y 530.977,Z 284.346,A -85,B 0,C 180,E1 -4303.07,E2 -4303.07} C_VEL
LIN {X 0,Y 531.043,Z 284.341,A -85,B 0,C 180,E1 -4305.436,E2 -4305.436} C_VEL
LIN {X 0,Y 531.039,Z 284.331,A -85,B 0,C 180,E1 -4308.55,E2 -4308.55} C_VEL
LIN {X 0,Y 531.05,Z 284.339,A -85,B 0,C 180,E1 -4311.629,E2 -4311.629} C_VEL
LIN {X 0,Y 531.119,Z 284.322,A -85,B 0,C 180,E1 -4314.685,E2 -4314.685} C_VEL
LIN {X 0,Y 531.139,Z 284.327,A -85,B 0,C 180,E1 -4317.725,E2 -4317.725} C_VEL
LIN {X 0,Y 531.152,Z 284.316,A -85,B 0,C 180,E1 -4320.758,E2 -4320.758} C_VEL
LIN {X 0,Y 531.105,Z 284.323,A -85,B 0,C 180,E1 -4323.034,E2 -4323.034} C_VEL
LIN {X 0,Y 531.069,Z 284.336,A -85,B 0,C 180,E1 -4326.077,E2 -4326.077} C_VEL
LIN {X 0,Y 531.054,Z 284.336,A -85,B 0,C 180,E1 -4328.37,E2 -4328.37} C_VEL
LIN {X 0,Y 531.053,Z 284.33,A -85,B 0,C 180,E1 -4331.672,E2 -4331.672} C_VEL
LIN {X 0,Y 531.033,Z 284.334,A -85,B 0,C 180,E1 -4334.956,E2 -4334.956} C_VEL
LIN {X 0,Y 530.982,Z 284.336,A -85,B 0,C 180,E1 -4337.723,E2 -4337.723} C_VEL
LIN {X 0,Y 531.026,Z 284.336,A -85,B 0,C 180,E1 -4340.127,E2 -4340.127} C_VEL
LIN {X 0,Y 530.946,Z 284.35,A -85,B 0,C 180,E1 -4342.573,E2 -4342.573} C_VEL
LIN {X 0,Y 531.006,Z 284.339,A -85,B 0,C 180,E1 -4345.057,E2 -4345.057} C_VEL
LIN {X 0,Y 531.014,Z 284.332,A -85,B 0,C 180,E1 -4347.596,E2 -4347.596} C_VEL
LIN {X 0,Y 530.976,Z 284.344,A -85,B 0,C 180,E1 -4350.645,E2 -4350.645} C_VEL
LIN {X 0,Y 530.956,Z 284.341,A -85,B 0,C 180,E1 -4353.775,E2 -4353.775} C_VEL
LIN {X 0,Y 530.956,Z 284.343,A -85,B 0,C 180,E1 -4356.558,E2 -4356.558} C_VEL
LIN {X 0,Y 530.987,Z 284.343,A -85,B 0,C 180,E1 -4359.443,E2 -4359.443} C_VEL
LIN {X 0,Y 530.979,Z 284.339,A -85,B 0,C 180,E1 -4362.457,E2 -4362.457} C_VEL
LIN {X 0,Y 530.978,Z 284.345,A -85,B 0,C 180,E1 -4365.622,E2 -4365.622} C_VEL
LIN {X 0,Y 530.995,Z 284.336,A -85,B 0,C 180,E1 -4368.564,E2 -4368.564} C_VEL
LIN {X 0,Y 530.959,Z 284.351,A -85,B 0,C 180,E1 -4371.529,E2 -4371.529} C_VEL
LIN {X 0,Y 530.956,Z 284.344,A -85,B 0,C 180,E1 -4374.38,E2 -4374.38} C_VEL
LIN {X 0,Y 530.969,Z 284.344,A -85,B 0,C 180,E1 -4377.133,E2 -4377.133} C_VEL
LIN {X 0,Y 530.973,Z 284.348,A -85,B 0,C 180,E1 -4379.803,E2 -4379.803} C_VEL
LIN {X 0,Y 531.013,Z 284.34,A -85,B 0,C 180,E1 -4382.468,E2 -4382.468} C_VEL
LIN {X 0,Y 531.005,Z 284.34,A -85,B 0,C 180,E1 -4384.942,E2 -4384.942} C_VEL
LIN {X 0,Y 531.012,Z 284.426,A -85,B 0,C 180,E1 -4385.808,E2 -4385.808} C_VEL
LIN {X 0,Y 532.225,Z 292.442,A -85,B 0,C 180,E1 -4387.073,E2 -4387.073} C_VEL
LIN {X 0,Y 531.87,Z 311.267,A -85,B 0,C 180,E1 -4389.906,E2 -4389.906} C_VEL
LIN {X 0,Y 531.498,Z 331.176,A -85,B 0,C 180,E1 -4392.889,E2 -4392.889} C_VEL
LIN {X 0,Y 531.303,Z 345.778,A -85,B 0,C 180,E1 -4395.048,E2 -4395.048} C_VEL
LIN {X 0,Y 532.751,Z 356.571,A -85,B 0,C 180,E1 -4395.242,E2 -4395.242} C_VEL
LIN {X 0,Y 532.328,Z 454.699,A -85,B 0,C 180,E1 -4396.593,E2 -4396.593} C_VEL
LIN {X 0,Y 532.189,Z 467.85,A -85,B 0,C 180,E1 -4396.929,E2 -4396.929} C_VEL
LIN {X 0,Y 531.955,Z 480.531,A -85,B 0,C 180,E1 -4397.409,E2 -4397.409} C_VEL
LIN {X 0,Y 531.746,Z 491.61,A -85,B 0,C 180,E1 -4397.973,E2 -4397.973} C_VEL
LIN {X 0,Y 531.493,Z 503.486,A -85,B 0,C 180,E1 -4398.753,E2 -4398.753} C_VEL
LIN {X 0,Y 531.203,Z 513.993,A -85,B 0,C 180,E1 -4399.615,E2 -4399.615} C_VEL
LIN {X 0,Y 531.019,Z 522.585,A -85,B 0,C 180,E1 -4400.477,E2 -4400.477} C_VEL
LIN {X 0,Y 530.842,Z 530.509,A -85,B 0,C 180,E1 -4401.434,E2 -4401.434} C_VEL
LIN {X 0,Y 530.675,Z 538.245,A -85,B 0,C 180,E1 -4402.581,E2 -4402.581} C_VEL
LIN {X 0,Y 530.588,Z 545.371,A -85,B 0,C 180,E1 -4403.917,E2 -4403.917} C_VEL
LIN {X 0,Y 530.459,Z 550.109,A -85,B 0,C 180,E1 -4405.059,E2 -4405.059} C_VEL
LIN {X 0,Y 530.516,Z 553.734,A -85,B 0,C 180,E1 -4406.202,E2 -4406.202} C_VEL
LIN {X 0,Y 530.457,Z 555.601,A -85,B 0,C 180,E1 -4406.962,E2 -4406.962} C_VEL
LIN {X 0,Y 530.41,Z 557,A -85,B 0,C 180,E1 -4407.721,E2 -4407.721} C_VEL
LIN {X 0,Y 530.344,Z 558.607,A -85,B 0,C 180,E1 -4409.24,E2 -4409.24} C_VEL
LIN {X 0,Y 530.345,Z 558.826,A -85,B 0,C 180,E1 -4410,E2 -4410} C_VEL
LIN {X 0,Y 530.36,Z 558.003,A -85,B 0,C 180,E1 -4411.518,E2 -4411.518} C_VEL
LIN {X 0,Y 530.41,Z 557.008,A -85,B 0,C 180,E1 -4412.278,E2 -4412.278} C_VEL
LIN {X 0,Y 530.457,Z 555.612,A -85,B 0,C 180,E1 -4413.037,E2 -4413.037} C_VEL
LIN {X 0,Y 530.522,Z 552.673,A -85,B 0,C 180,E1 -4414.178,E2 -4414.178} C_VEL
LIN {X 0,Y 530.524,Z 548.69,A -85,B 0,C 180,E1 -4415.32,E2 -4415.32} C_VEL
LIN {X 0,Y 530.594,Z 542.973,A -85,B 0,C 180,E1 -4416.578,E2 -4416.578} C_VEL
LIN {X 0,Y 530.719,Z 535.867,A -85,B 0,C 180,E1 -4417.801,E2 -4417.801} C_VEL
LIN {X 0,Y 530.909,Z 527.558,A -85,B 0,C 180,E1 -4418.948,E2 -4418.948} C_VEL
LIN {X 0,Y 531.102,Z 519.035,A -85,B 0,C 180,E1 -4419.905,E2 -4419.905} C_VEL
LIN {X 0,Y 531.358,Z 508.502,A -85,B 0,C 180,E1 -4420.863,E2 -4420.863} C_VEL
LIN {X 0,Y 531.605,Z 497.491,A -85,B 0,C 180,E1 -4421.67,E2 -4421.67} C_VEL
LIN {X 0,Y 531.863,Z 486.645,A -85,B 0,C 180,E1 -4422.302,E2 -4422.302} C_VEL
LIN {X 0,Y 532.04,Z 474.861,A -85,B 0,C 180,E1 -4422.831,E2 -4422.831} C_VEL
LIN {X 0,Y 532.278,Z 461.279,A -85,B 0,C 180,E1 -4423.262,E2 -4423.262} C_VEL
LIN {X 0,Y 532.414,Z 449.244,A -85,B 0,C 180,E1 -4423.501,E2 -4423.501} C_VEL
LIN {X 0,Y 532.628,Z 354.634,A -85,B 0,C 180,E1 -4424.791,E2 -4424.791} C_VEL
LIN {X 0,Y 531.312,Z 345.957,A -85,B 0,C 180,E1 -4424.966,E2 -4424.966} C_VEL
LIN {X 0,Y 531.718,Z 325.065,A -85,B 0,C 180,E1 -4428.117,E2 -4428.117} C_VEL
LIN {X 0,Y 532.066,Z 306.844,A -85,B 0,C 180,E1 -4430.893,E2 -4430.893} C_VEL
LIN {X 0,Y 532.423,Z 292.487,A -85,B 0,C 180,E1 -4433.122,E2 -4433.122} C_VEL
LIN {X 0,Y 530.996,Z 284.343,A -85,B 0,C 180,E1 -4434.483,E2 -4434.483} C_VEL
LIN {X 0,Y 531.015,Z 284.339,A -85,B 0,C 180,E1 -4437.532,E2 -4437.532} C_VEL
LIN {X 0,Y 530.973,Z 284.341,A -85,B 0,C 180,E1 -4440.644,E2 -4440.644} C_VEL
LIN {X 0,Y 530.986,Z 284.34,A -85,B 0,C 180,E1 -4443.772,E2 -4443.772} C_VEL
LIN {X 0,Y 530.953,Z 284.346,A -85,B 0,C 180,E1 -4446.558,E2 -4446.558} C_VEL
LIN {X 0,Y 530.983,Z 284.337,A -85,B 0,C 180,E1 -4449.443,E2 -4449.443} C_VEL
LIN {X 0,Y 530.977,Z 284.348,A -85,B 0,C 180,E1 -4452.456,E2 -4452.456} C_VEL
LIN {X 0,Y 530.984,Z 284.337,A -85,B 0,C 180,E1 -4455.62,E2 -4455.62} C_VEL
LIN {X 0,Y 530.997,Z 284.346,A -85,B 0,C 180,E1 -4458.565,E2 -4458.565} C_VEL
LIN {X 0,Y 530.955,Z 284.341,A -85,B 0,C 180,E1 -4461.529,E2 -4461.529} C_VEL
LIN {X 0,Y 530.972,Z 284.343,A -85,B 0,C 180,E1 -4464.381,E2 -4464.381} C_VEL
LIN {X 0,Y 530.968,Z 284.344,A -85,B 0,C 180,E1 -4467.133,E2 -4467.133} C_VEL
LIN {X 0,Y 530.965,Z 284.34,A -85,B 0,C 180,E1 -4469.803,E2 -4469.803} C_VEL
LIN {X 0,Y 531.01,Z 284.336,A -85,B 0,C 180,E1 -4472.467,E2 -4472.467} C_VEL
LIN {X 0,Y 531.001,Z 284.344,A -85,B 0,C 180,E1 -4474.942,E2 -4474.942} C_VEL
LIN {X 0,Y 530.966,Z 284.339,A -85,B 0,C 180,E1 -4478.246,E2 -4478.246} C_VEL
LIN {X 0,Y 530.99,Z 284.339,A -85,B 0,C 180,E1 -4480.677,E2 -4480.677} C_VEL
LIN {X 0,Y 530.98,Z 284.345,A -85,B 0,C 180,E1 -4483.071,E2 -4483.071} C_VEL
LIN {X 0,Y 531.035,Z 284.339,A -85,B 0,C 180,E1 -4485.436,E2 -4485.436} C_VEL
LIN {X 0,Y 531.03,Z 284.331,A -85,B 0,C 180,E1 -4488.55,E2 -4488.55} C_VEL
LIN {X 0,Y 531.051,Z 284.337,A -85,B 0,C 180,E1 -4491.63,E2 -4491.63} C_VEL
LIN {X 0,Y 531.116,Z 284.321,A -85,B 0,C 180,E1 -4494.685,E2 -4494.685} C_VEL
LIN {X 0,Y 531.131,Z 284.328,A -85,B 0,C 180,E1 -4497.725,E2 -4497.725} C_VEL
LIN {X 0,Y 531.145,Z 284.317,A -85,B 0,C 180,E1 -4500.758,E2 -4500.758} C_VEL
LIN {X 0,Y 531.099,Z 284.323,A -85,B 0,C 180,E1 -4503.034,E2 -4503.034} C_VEL
LIN {X 0,Y 531.065,Z 284.334,A -85,B 0,C 180,E1 -4506.078,E2 -4506.078} C_VEL
LIN {X 0,Y 531.05,Z 284.332,A -85,B 0,C 180,E1 -4508.371,E2 -4508.371} C_VEL
LIN {X 0,Y 531.045,Z 284.334,A -85,B 0,C 180,E1 -4511.672,E2 -4511.672} C_VEL
LIN {X 0,Y 531.024,Z 284.332,A -85,B 0,C 180,E1 -4514.956,E2 -4514.956} C_VEL
LIN {X 0,Y 530.975,Z 284.341,A -85,B 0,C 180,E1 -4517.724,E2 -4517.724} C_VEL
LIN {X 0,Y 531.019,Z 284.34,A -85,B 0,C 180,E1 -4520.128,E2 -4520.128} C_VEL
LIN {X 0,Y 530.94,Z 284.349,A -85,B 0,C 180,E1 -4522.574,E2 -4522.574} C_VEL
LIN {X 0,Y 530.984,Z 284.338,A -85,B 0,C 180,E1 -4525.059,E2 -4525.059} C_VEL
LIN {X 0,Y 530.965,Z 284.34,A -85,B 0,C 180,E1 -4527.599,E2 -4527.599} C_VEL
LIN {X 0,Y 530.964,Z 284.344,A -85,B 0,C 180,E1 -4530.198,E2 -4530.198} C_VEL
LIN {X 0,Y 530.963,Z 284.346,A -85,B 0,C 180,E1 -4532.867,E2 -4532.867} C_VEL
LIN {X 0,Y 530.95,Z 284.341,A -85,B 0,C 180,E1 -4535.621,E2 -4535.621} C_VEL
LIN {X 0,Y 530.962,Z 284.348,A -85,B 0,C 180,E1 -4538.654,E2 -4538.654} C_VEL
LIN {X 0,Y 530.983,Z 284.339,A -85,B 0,C 180,E1 -4541.437,E2 -4541.437} C_VEL
LIN {X 0,Y 530.934,Z 284.345,A -85,B 0,C 180,E1 -4543.546,E2 -4543.546} C_VEL
LIN {X 0,Y 530.268,Z 284.427,A -85,B 0,C 180,E1 -4544.18,E2 -4544.18} C_VEL
LIN {X 0,Y 527.43,Z 284.787,A -85,B 0,C 180,E1 -4545.209,E2 -4545.209} C_VEL
LIN {X 0,Y 525.026,Z 285.09,A -85,B 0,C 180,E1 -4546.038,E2 -4546.038} C_VEL
LIN {X 0,Y 523.984,Z 285.218,A -85,B 0,C 180,E1 -4546.677,E2 -4546.677} C_VEL
LIN {X 0,Y 523.894,Z 285.227,A -85,B 0,C 180,E1 -4546.894,E2 -4546.894} C_VEL
LIN {X 0,Y 523.911,Z 285.218,A -85,B 0,C 180,E1 -4549.918,E2 -4549.918} C_VEL
LIN {X 0,Y 523.904,Z 285.224,A -85,B 0,C 180,E1 -4552.868,E2 -4552.868} C_VEL
LIN {X 0,Y 523.919,Z 285.22,A -85,B 0,C 180,E1 -4555.71,E2 -4555.71} C_VEL
LIN {X 0,Y 523.911,Z 285.218,A -85,B 0,C 180,E1 -4558.456,E2 -4558.456} C_VEL
LIN {X 0,Y 523.906,Z 285.225,A -85,B 0,C 180,E1 -4561.124,E2 -4561.124} C_VEL
LIN {X 0,Y 523.895,Z 285.222,A -85,B 0,C 180,E1 -4564.002,E2 -4564.002} C_VEL
LIN {X 0,Y 523.91,Z 285.219,A -85,B 0,C 180,E1 -4566.27,E2 -4566.27} C_VEL
LIN {X 0,Y 523.947,Z 285.214,A -85,B 0,C 180,E1 -4568.767,E2 -4568.767} C_VEL
LIN {X 0,Y 523.921,Z 285.22,A -85,B 0,C 180,E1 -4571.22,E2 -4571.22} C_VEL
LIN {X 0,Y 523.907,Z 285.227,A -85,B 0,C 180,E1 -4573.639,E2 -4573.639} C_VEL
LIN {X 0,Y 523.932,Z 285.222,A -85,B 0,C 180,E1 -4576.028,E2 -4576.028} C_VEL
LIN {X 0,Y 523.963,Z 285.214,A -85,B 0,C 180,E1 -4578.394,E2 -4578.394} C_VEL
LIN {X 0,Y 523.949,Z 285.217,A -85,B 0,C 180,E1 -4581.516,E2 -4581.516} C_VEL
LIN {X 0,Y 524.032,Z 285.205,A -85,B 0,C 180,E1 -4584.614,E2 -4584.614} C_VEL
LIN {X 0,Y 524.103,Z 285.198,A -85,B 0,C 180,E1 -4587.695,E2 -4587.695} C_VEL
LIN {X 0,Y 524.099,Z 285.202,A -85,B 0,C 180,E1 -4590,E2 -4590} C_VEL
LIN {X 0,Y 524.101,Z 285.204,A -85,B 0,C 180,E1 -4592.306,E2 -4592.306} C_VEL
LIN {X 0,Y 524.006,Z 285.213,A -85,B 0,C 180,E1 -4596.16,E2 -4596.16} C_VEL
LIN {X 0,Y 523.941,Z 285.215,A -85,B 0,C 180,E1 -4599.263,E2 -4599.263} C_VEL
LIN {X 0,Y 523.921,Z 285.225,A -85,B 0,C 180,E1 -4602.394,E2 -4602.394} C_VEL
LIN {X 0,Y 523.888,Z 285.221,A -85,B 0,C 180,E1 -4605.564,E2 -4605.564} C_VEL
LIN {X 0,Y 523.915,Z 285.219,A -85,B 0,C 180,E1 -4607.971,E2 -4607.971} C_VEL
LIN {X 0,Y 523.926,Z 285.221,A -85,B 0,C 180,E1 -4610.412,E2 -4610.412} C_VEL
LIN {X 0,Y 523.894,Z 285.23,A -85,B 0,C 180,E1 -4612.895,E2 -4612.895} C_VEL
LIN {X 0,Y 523.865,Z 285.23,A -85,B 0,C 180,E1 -4615.424,E2 -4615.424} C_VEL
LIN {X 0,Y 523.967,Z 285.378,A -85,B 0,C 180,E1 -4617.267,E2 -4617.267} C_VEL
LIN {X 0,Y 524.519,Z 289.975,A -85,B 0,C 180,E1 -4618.185,E2 -4618.185} C_VEL
LIN {X 0,Y 524.257,Z 305.325,A -85,B 0,C 180,E1 -4621.146,E2 -4621.146} C_VEL
LIN {X 0,Y 524.203,Z 309.264,A -85,B 0,C 180,E1 -4621.892,E2 -4621.892} C_VEL
LIN {X 0,Y 525.946,Z 319.907,A -85,B 0,C 180,E1 -4622.113,E2 -4622.113} C_VEL
LIN {X 0,Y 525.509,Z 416.717,A -85,B 0,C 180,E1 -4623.473,E2 -4623.473} C_VEL
LIN {X 0,Y 525.299,Z 429.684,A -85,B 0,C 180,E1 -4623.812,E2 -4623.812} C_VEL
LIN {X 0,Y 525.1,Z 441.316,A -85,B 0,C 180,E1 -4624.262,E2 -4624.262} C_VEL
LIN {X 0,Y 524.836,Z 452.007,A -85,B 0,C 180,E1 -4624.805,E2 -4624.805} C_VEL
LIN {X 0,Y 524.619,Z 461.154,A -85,B 0,C 180,E1 -4625.384,E2 -4625.384} C_VEL
LIN {X 0,Y 524.376,Z 470.878,A -85,B 0,C 180,E1 -4626.137,E2 -4626.137} C_VEL
LIN {X 0,Y 524.163,Z 479.398,A -85,B 0,C 180,E1 -4626.934,E2 -4626.934} C_VEL
LIN {X 0,Y 523.978,Z 487.645,A -85,B 0,C 180,E1 -4627.861,E2 -4627.861} C_VEL
LIN {X 0,Y 523.774,Z 493.949,A -85,B 0,C 180,E1 -4628.704,E2 -4628.704} C_VEL
LIN {X 0,Y 523.619,Z 500.967,A -85,B 0,C 180,E1 -4629.833,E2 -4629.833} C_VEL
LIN {X 0,Y 523.509,Z 506.243,A -85,B 0,C 180,E1 -4630.879,E2 -4630.879} C_VEL
LIN {X 0,Y 523.416,Z 511.433,A -85,B 0,C 180,E1 -4632.172,E2 -4632.172} C_VEL
LIN {X 0,Y 523.344,Z 515.379,A -85,B 0,C 180,E1 -4633.517,E2 -4633.517} C_VEL
LIN {X 0,Y 523.329,Z 517.61,A -85,B 0,C 180,E1 -4634.621,E2 -4634.621} C_VEL
LIN {X 0,Y 523.297,Z 518.958,A -85,B 0,C 180,E1 -4635.703,E2 -4635.703} C_VEL
LIN {X 0,Y 523.256,Z 519.52,A -85,B 0,C 180,E1 -4636.764,E2 -4636.764} C_VEL
LIN {X 0,Y 523.299,Z 519.328,A -85,B 0,C 180,E1 -4637.816,E2 -4637.816} C_VEL
LIN {X 0,Y 523.306,Z 518.437,A -85,B 0,C 180,E1 -4638.847,E2 -4638.847} C_VEL
LIN {X 0,Y 523.327,Z 515.769,A -85,B 0,C 180,E1 -4640.411,E2 -4640.411} C_VEL
LIN {X 0,Y 523.414,Z 511.695,A -85,B 0,C 180,E1 -4641.855,E2 -4641.855} C_VEL
LIN {X 0,Y 523.504,Z 507.019,A -85,B 0,C 180,E1 -4643.053,E2 -4643.053} C_VEL
LIN {X 0,Y 523.627,Z 500.891,A -85,B 0,C 180,E1 -4644.278,E2 -4644.278} C_VEL
LIN {X 0,Y 523.761,Z 494.428,A -85,B 0,C 180,E1 -4645.324,E2 -4645.324} C_VEL
LIN {X 0,Y 523.969,Z 487.415,A -85,B 0,C 180,E1 -4646.264,E2 -4646.264} C_VEL
LIN {X 0,Y 524.233,Z 478.742,A -85,B 0,C 180,E1 -4647.229,E2 -4647.229} C_VEL
LIN {X 0,Y 524.44,Z 468.6,A -85,B 0,C 180,E1 -4648.152,E2 -4648.152} C_VEL
LIN {X 0,Y 524.753,Z 456.87,A -85,B 0,C 180,E1 -4648.998,E2 -4648.998} C_VEL
LIN {X 0,Y 524.986,Z 445.344,A -85,B 0,C 180,E1 -4649.644,E2 -4649.644} C_VEL
LIN {X 0,Y 525.248,Z 433.115,A -85,B 0,C 180,E1 -4650.159,E2 -4650.159} C_VEL
LIN {X 0,Y 525.334,Z 421.694,A -85,B 0,C 180,E1 -4650.506,E2 -4650.506} C_VEL
LIN {X 0,Y 525.511,Z 408.432,A -85,B 0,C 180,E1 -4650.754,E2 -4650.754} C_VEL
LIN {X 0,Y 525.863,Z 318.44,A -85,B 0,C 180,E1 -4652.003,E2 -4652.003} C_VEL
LIN {X 0,Y 524.181,Z 308.716,A -85,B 0,C 180,E1 -4652.211,E2 -4652.211} C_VEL
LIN {X 0,Y 524.184,Z 290.77,A -85,B 0,C 180,E1 -4655.229,E2 -4655.229} C_VEL
LIN {X 0,Y 524.039,Z 285.209,A -85,B 0,C 180,E1 -4656.162,E2 -4656.162} C_VEL
LIN {X 0,Y 523.974,Z 285.218,A -85,B 0,C 180,E1 -4659.59,E2 -4659.59} C_VEL
LIN {X 0,Y 523.96,Z 285.218,A -85,B 0,C 180,E1 -4662.837,E2 -4662.837} C_VEL
LIN {X 0,Y 524.007,Z 285.216,A -85,B 0,C 180,E1 -4665.236,E2 -4665.236} C_VEL
LIN {X 0,Y 524.015,Z 285.207,A -85,B 0,C 180,E1 -4668.394,E2 -4668.394} C_VEL
LIN {X 0,Y 523.998,Z 285.216,A -85,B 0,C 180,E1 -4671.516,E2 -4671.516} C_VEL
LIN {X 0,Y 524.08,Z 285.199,A -85,B 0,C 180,E1 -4674.613,E2 -4674.613} C_VEL
LIN {X 0,Y 524.111,Z 285.202,A -85,B 0,C 180,E1 -4677.694,E2 -4677.694} C_VEL
LIN {X 0,Y 524.123,Z 285.191,A -85,B 0,C 180,E1 -4680.768,E2 -4680.768} C_VEL
LIN {X 0,Y 524.072,Z 285.199,A -85,B 0,C 180,E1 -4683.075,E2 -4683.075} C_VEL
LIN {X 0,Y 524.027,Z 285.212,A -85,B 0,C 180,E1 -4686.159,E2 -4686.159} C_VEL
LIN {X 0,Y 524.002,Z 285.213,A -85,B 0,C 180,E1 -4688.484,E2 -4688.484} C_VEL
LIN {X 0,Y 524.004,Z 285.209,A -85,B 0,C 180,E1 -4691.739,E2 -4691.739} C_VEL
LIN {X 0,Y 523.996,Z 285.21,A -85,B 0,C 180,E1 -4695.053,E2 -4695.053} C_VEL
LIN {X 0,Y 523.949,Z 285.214,A -85,B 0,C 180,E1 -4697.969,E2 -4697.969} C_VEL
LIN {X 0,Y 523.973,Z 285.218,A -85,B 0,C 180,E1 -4700.41,E2 -4700.41} C_VEL
LIN {X 0,Y 523.912,Z 285.224,A -85,B 0,C 180,E1 -4702.893,E2 -4702.893} C_VEL
LIN {X 0,Y 523.954,Z 285.214,A -85,B 0,C 180,E1 -4705.419,E2 -4705.419} C_VEL
LIN {X 0,Y 523.969,Z 285.21,A -85,B 0,C 180,E1 -4707.999,E2 -4707.999} C_VEL
LIN {X 0,Y 523.946,Z 285.223,A -85,B 0,C 180,E1 -4710.855,E2 -4710.855} C_VEL
LIN {X 0,Y 523.931,Z 285.217,A -85,B 0,C 180,E1 -4713.729,E2 -4713.729} C_VEL
LIN {X 0,Y 523.905,Z 285.221,A -85,B 0,C 180,E1 -4716.401,E2 -4716.401} C_VEL
LIN {X 0,Y 523.922,Z 285.225,A -85,B 0,C 180,E1 -4719.085,E2 -4719.085} C_VEL
LIN {X 0,Y 523.953,Z 285.215,A -85,B 0,C 180,E1 -4722.119,E2 -4722.119} C_VEL
LIN {X 0,Y 523.944,Z 285.224,A -85,B 0,C 180,E1 -4725.31,E2 -4725.31} C_VEL
LIN {X 0,Y 523.958,Z 285.213,A -85,B 0,C 180,E1 -4728.69,E2 -4728.69} C_VEL
LIN {X 0,Y 523.919,Z 285.221,A -85,B 0,C 180,E1 -4731.081,E2 -4731.081} C_VEL
LIN {X 0,Y 523.903,Z 285.23,A -85,B 0,C 180,E1 -4733.825,E2 -4733.825} C_VEL
LIN {X 0,Y 523.944,Z 285.218,A -85,B 0,C 180,E1 -4736.635,E2 -4736.635} C_VEL
LIN {X 0,Y 523.959,Z 285.218,A -85,B 0,C 180,E1 -4739.356,E2 -4739.356} C_VEL
LIN {X 0,Y 523.978,Z 285.218,A -85,B 0,C 180,E1 -4742.282,E2 -4742.282} C_VEL
LIN {X 0,Y 523.953,Z 285.221,A -85,B 0,C 180,E1 -4744.581,E2 -4744.581} C_VEL
LIN {X 0,Y 523.969,Z 285.403,A -85,B 0,C 180,E1 -4745.68,E2 -4745.68} C_VEL
LIN {X 0,Y 525.246,Z 293.345,A -85,B 0,C 180,E1 -4746.96,E2 -4746.96} C_VEL
LIN {X 0,Y 524.893,Z 312.246,A -85,B 0,C 180,E1 -4749.832,E2 -4749.832} C_VEL
LIN {X 0,Y 524.532,Z 330.877,A -85,B 0,C 180,E1 -4752.655,E2 -4752.655} C_VEL
LIN {X 0,Y 524.294,Z 345.619,A -85,B 0,C 180,E1 -4754.847,E2 -4754.847} C_VEL
LIN {X 0,Y 525.9,Z 357.368,A -85,B 0,C 180,E1 -4755.061,E2 -4755.061} C_VEL
LIN {X 0,Y 525.427,Z 454.143,A -85,B 0,C 180,E1 -4756.413,E2 -4756.413} C_VEL
LIN {X 0,Y 525.28,Z 467.379,A -85,B 0,C 180,E1 -4756.754,E2 -4756.754} C_VEL
LIN {X 0,Y 524.997,Z 480.105,A -85,B 0,C 180,E1 -4757.239,E2 -4757.239} C_VEL
LIN {X 0,Y 524.755,Z 492.259,A -85,B 0,C 180,E1 -4757.874,E2 -4757.874} C_VEL
LIN {X 0,Y 524.475,Z 504.426,A -85,B 0,C 180,E1 -4758.698,E2 -4758.698} C_VEL
LIN {X 0,Y 524.152,Z 514.711,A -85,B 0,C 180,E1 -4759.571,E2 -4759.571} C_VEL
LIN {X 0,Y 523.945,Z 523.953,A -85,B 0,C 180,E1 -4760.542,E2 -4760.542} C_VEL
LIN {X 0,Y 523.729,Z 532.95,A -85,B 0,C 180,E1 -4761.705,E2 -4761.705} C_VEL
LIN {X 0,Y 523.573,Z 540.194,A -85,B 0,C 180,E1 -4762.867,E2 -4762.867} C_VEL
